Universal Robots PolyScope program: Cover LT.urp

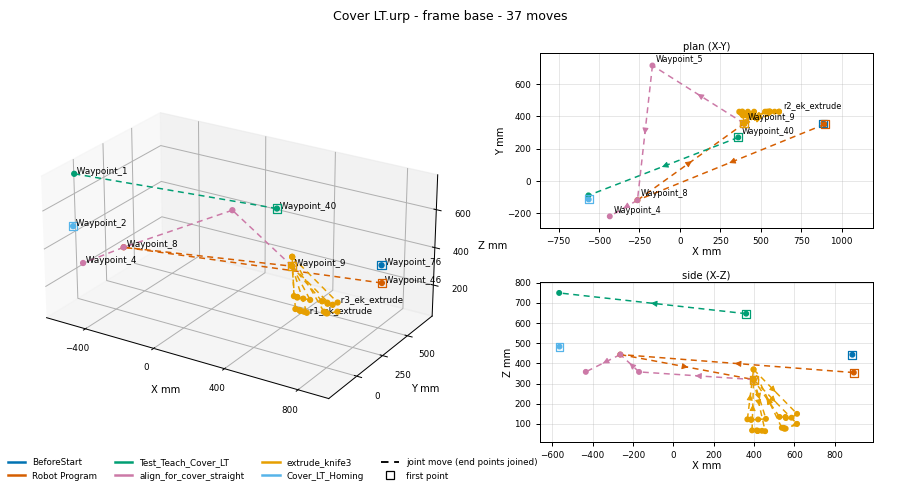
[picture p0: tool path of Cover LT.urp in frame base, 37 of 60 moves have a stored position in this frame; points joined in program order, loops and branches not executed]
Program Cover LT (installation=robot2 directory=/programs/UPF createdIn=5.14.5 lastSavedIn=5.21.3 robotSerialNumber=20246801938)
Calibrated DH parameters: a=[-0.000071, -0.790281, -0.600694, 0.000061, -0.000039, 0]; d=[0.236272, 604.465945, 132.116513, -736.382239, 0.159268, 0.154005]; alpha=[1.570254, -0.000567, 0.000559, 1.571709, -1.56999, 0]; deltaTheta=[0, -0.409357, 7.293326, -0.600784, -0.000001, -0.000001]
InitVariablesNode variables(variable(name=free_dr_already, expression=False), variable(name=freedrive_m_var, expression=False))
BeforeStart
  SuppressedNode
    Folder Safe Home Folder
      'if robot is not at home, send it back to home safely'
      'make sure the tcp is welder'
      Set NoAction tcp=pretend_welder
      sp := get_actual_tcp_pose()
      MoveL speed 250 mm/s, acceleration 1200 mm/s^2 (useActiveTCP=true optimoveEnabled=false optiMoveSpeed=0.3 optiMoveAcceleration=0.09) feature=Base
        Waypoint Variable (Variable): variable=sp
        'if first move is to a variable, skip automove'
      'turn off welder'
      URCap WireTank Serial (WireTank Serial, WireTank, LLC) dataModel(NODE_TITLE=Serial Bridge uR0, Command=[252,82,48], QUERY=false, byte_array=true, OUTPUT_ENTRY=Static, Variable(key=OUTPUT_VARIABLE, variable(name=HwResp)))
      Set DigitalOutput pin=digital_out[0]; digitalValue=0
      jp := get_actual_joint_positions()
      If sp[0]>0.600
        'if x > 600 then above then home'
        MoveJ speed 60 deg/s, acceleration 80 deg/s^2 (useActiveTCP=true optimoveEnabled=false optiMoveSpeed=0.3 optiMoveAcceleration=0.09) feature=Base
          SuppressedNode
            Waypoint Waypoint_47: TCP in base x=894.111 y=351.078 z=354.441 mm, rx=2.3264 ry=2.0525 rz=0.0574 rad; joints [-187.182, -67.293, 94.726, 57.522, -0.141, -88.018] deg; TCP offset x=-5.49 y=-328 z=106.39 mm, rx=1.2092 ry=-1.2092 rz=1.2092 rad
          Waypoint Waypoint_76: TCP in base x=886.939 y=356.263 z=442.999 mm, rx=2.3163 ry=2.0576 rz=0.0741 rad; joints [-187.059, -71.746, 90.665, 52.573, -0.48, -75.13] deg; TCP offset x=-9.5 y=-328 z=105.73 mm, rx=1.2092 ry=-1.2092 rz=1.2092 rad
        SafeHome (positionOptionType=SPEED_AND_ACCELERATION speed=1.047198 acceleration=1.396263 nextMotionTime=2)
      Else 
        Popup Message (haltProgram=false message=retreating to home inputType=Text)
        'for rules 2-8, finish with oldhome then above then home'
        If -1.74<jp[4] and jp[4]<1.05 and -1.74<jp[3] and jp[3]<1.74
          'if oldhome, test teach, then go straight to oldhome'
        ElseIf sp[0]<-.5 and jp[3]>3.14 and -2.62<jp[4] and jp[4]<-0.87
          'if left side weld approach, left weld approach in reverse'
          MoveJ speed 60 deg/s, acceleration 80 deg/s^2 (useActiveTCP=true optimoveEnabled=false optiMoveSpeed=0.3 optiMoveAcceleration=0.09) feature=Base
            Waypoint Waypoint_50: TCP in base x=-568.711 y=230.602 z=220.209 mm, rx=-1.5191 ry=-0.5351 rz=0.574 rad; joints [-1.233, -73.308, 139.365, 291.685, -131.758, 87.871] deg; TCP offset x=-5.49 y=-328 z=106.39 mm, rx=1.2092 ry=-1.2092 rz=1.2092 rad
            Waypoint Waypoint_51: TCP in base x=-689.65 y=139.001 z=230.693 mm, rx=-0.852 ry=-1.646 rz=1.646 rad; joints [-65.631, -88.39, 163.033, 285.278, -280.919, 90.062] deg
            Waypoint Waypoint_52: TCP in base x=-160.992 y=970.528 z=722.037 mm, rx=-0.555 ry=0.1065 rz=0.3285 rad; joints [-74.362, -75.728, 129.393, 212.138, -169.184, 55.164] deg
            Waypoint Waypoint_53: TCP in base x=-157.624 y=513.351 z=815.67 mm, rx=-0.6727 ry=-1.8523 rz=-0.0554 rad; joints [-158.576, -104.315, 132.512, 57.998, -61.68, -46.426] deg
        ElseIf sp[0]<0 and 0<jp[3] and jp[3]<1.74 and 0.87<jp[4] and jp[4]<2.62
          'if right side around, move back then wapoint 24 then oldhome'
          If sp[0]<-1.0
            xback := p[-1.0,sp[1],sp[2],sp[3],sp[4],sp[5]]
            MoveJ speed 60 deg/s, acceleration 80 deg/s^2 (useActiveTCP=true optimoveEnabled=false optiMoveSpeed=0.3 optiMoveAcceleration=0.09) feature=Base
              Waypoint Variable (Variable): variable=xback
          MoveJ speed 60 deg/s, acceleration 80 deg/s^2 (useActiveTCP=true optimoveEnabled=false optiMoveSpeed=0.3 optiMoveAcceleration=0.09) feature=Base
            Waypoint Waypoint_54: TCP in base x=-308.528 y=606.081 z=242.371 mm, rx=-2.1337 ry=0.3494 rz=2.131 rad; joints [-112.4, -74.451, 126.505, 42.726, 91.418, 81.282] deg
        ElseIf jp[3]>2.62 and jp[4]<-3.84
          'if left side second half, then left weld ending sequence'
          If jp[5]<0.35
            MoveJ speed 60 deg/s, acceleration 80 deg/s^2 (useActiveTCP=true optimoveEnabled=false optiMoveSpeed=0.3 optiMoveAcceleration=0.09) feature=Base
              Waypoint Waypoint_65: TCP in base x=-850.3 y=-229.061 z=580.194 mm, rx=-0.0667 ry=-1.5664 rz=-0.0455 rad; joints [6.605, -69.14, 152.414, 186.359, -269.256, -10.612] deg
          MoveJ speed 60 deg/s, acceleration 80 deg/s^2 (useActiveTCP=true optimoveEnabled=false optiMoveSpeed=0.3 optiMoveAcceleration=0.09) feature=Base
            SuppressedNode
              Waypoint Waypoint_61: TCP in base x=-1224.453 y=315.135 z=45.036 mm, rx=0.4556 ry=-1.5209 rz=0.4778 rad; joints [-38.105, -18.537, 102.715, 186.465, -269.531, 72.317] deg
            SuppressedNode
              Waypoint Waypoint_62: TCP in base x=-1246.058 y=121.907 z=25.888 mm, rx=-0.7807 ry=-1.4195 rz=-0.7637 rad; joints [-2.239, -16.844, 100.196, 185.863, -269.635, -54.527] deg
            SuppressedNode
              Waypoint Waypoint_63: TCP in base x=-850.3 y=142.696 z=580.194 mm, rx=-0.0667 ry=-1.5664 rz=-0.0455 rad; joints [-33.715, -70.118, 156.539, 183.763, -269.222, 29.711] deg
            SuppressedNode
              Waypoint Waypoint_64: TCP in base x=-850.307 y=-229.065 z=580.197 mm, rx=-0.0667 ry=-1.5664 rz=-0.0455 rad; joints [6.605, -69.141, 152.414, 186.36, -269.255, -10.612] deg
            'above is testing, below is real'
            Waypoint Waypoint_55: TCP in base x=-850.296 y=369.354 z=580.191 mm, rx=-0.0667 ry=-1.5664 rz=-0.0455 rad; joints [-51.358, -68.674, 149.321, 189.759, -269.326, 47.358] deg
            SuppressedNode
              Waypoint Waypoint_60: TCP in base x=-826.865 y=369.366 z=43.112 mm, rx=0.575 ry=-1.4922 rz=0.5971 rad; joints [-59.177, -17.074, 121.534, 166.294, -269.929, 102.173] deg
            Waypoint Waypoint_59: motionParameters(nextMotionTime=2); TCP in base x=-689.651 y=138.973 z=230.7 mm, rx=-0.852 ry=-1.646 rz=1.646 rad; joints [-65.63, -88.392, 163.034, 285.278, -280.919, 90.062] deg
            Waypoint Waypoint_71: TCP in base x=-289.685 y=534.258 z=757.199 mm, rx=-0.2952 ry=-0.653 rz=0.3894 rad; joints [-79.881, -94.829, 156.624, 238.16, -217.621, 99.184] deg
            Waypoint Waypoint_58: TCP in base x=191.12 y=567.518 z=815.513 mm, rx=-0.1358 ry=0.3961 rz=0.2088 rad; joints [-94.611, -101.484, 149.999, 189.458, -152.19, 49.064] deg
            Waypoint Waypoint_56: TCP in base x=-254.568 y=502.959 z=1135.401 mm, rx=-0.2619 ry=-0.7497 rz=1.3491 rad; joints [-116.567, -108.934, 141.5, 126.12, -66.905, -29.189] deg
            Waypoint Waypoint_57: TCP in base x=-9.221 y=593.713 z=505.809 mm, rx=-1.4244 ry=-2.3441 rz=-0.5276 rad; joints [-167.352, -114.202, 136.688, 39.052, -32.592, -65.93] deg
        ElseIf jp[3]<-2.09
          'bottom homing'
          MoveJ speed 60 deg/s, acceleration 80 deg/s^2 (useActiveTCP=true optimoveEnabled=false optiMoveSpeed=0.3 optiMoveAcceleration=0.09) feature=Base
            SuppressedNode
              Waypoint Waypoint_66: TCP in base x=-1189.333 y=-102.843 z=-176.058 mm, rx=1.1963 ry=-1.1853 rz=1.2301 rad; joints [-19.887, -1.876, 78.341, -165.92, 91.498, 110.543] deg
            ''
            If sp[0]<-0.95
              xback := p[-0.95,sp[1],sp[2],sp[3],sp[4],sp[5]]
              MoveL speed 250 mm/s, acceleration 1200 mm/s^2 (useActiveTCP=true optimoveEnabled=false optiMoveSpeed=0.3 optiMoveAcceleration=0.09) feature=Base
                Waypoint Variable (Variable): variable=xback
            Waypoint Waypoint_67: TCP in base x=-339.169 y=114.271 z=51.007 mm, rx=-0.4342 ry=1.8727 rz=-1.8852 rad; joints [-80.817, -56.025, 141.954, -98.756, -22.671, 103.625] deg
        ElseIf jp[3]<0 and jp[4]<-3.14
          'if left side homing, special unspin'
          MoveJ speed 60 deg/s, acceleration 80 deg/s^2 (useActiveTCP=true optimoveEnabled=false optiMoveSpeed=0.3 optiMoveAcceleration=0.09) feature=Base
            SuppressedNode
              Waypoint Waypoint_68: TCP in base x=-1436.144 y=-207.487 z=20.65 mm, rx=-1.0168 ry=-1.7024 rz=1.6295 rad; joints [2.271, -43.137, 96.498, -42.2, -211.884, 93.908] deg
            ''
            Waypoint Waypoint_69: TCP in base x=-760.827 y=-49.763 z=82.65 mm, rx=-1.0262 ry=-1.6127 rz=1.5471 rad; joints [-12.694, -64.084, 157.914, -89.201, -220.703, 89.352] deg
            Waypoint Waypoint_70: TCP in base x=-154.415 y=636.923 z=16.979 mm, rx=-0.3028 ry=1.487 rz=0.1222 rad; joints [-64.641, -61.184, 139.176, -160.395, -91.873, 99.702] deg
        ElseIf (sp[4]<-3 or sp[4]>3) and -0.02<sp[5] and sp[5]<0.02
          'go straight to home'
        ElseIf 2>1
          'if none of the other options, then error continuously'
          Loop While (checkContinuously=false) expression=2>1
            Popup Message (haltProgram=false message=Unknown Position. Find Calvin for Assistance inputType=Text)
        'insert logic for how to get back to oldhome'
        'finish with oldhome then above then home'
        MoveJ speed 60 deg/s, acceleration 80 deg/s^2 (useActiveTCP=true optimoveEnabled=false optiMoveSpeed=0.3 optiMoveAcceleration=0.09) feature=Base
          Waypoint Waypoint_49: motionParameters(jointSpeed=1.047198 jointAcceleration=1.396263 cartesianSpeed=0.25 cartesianAcceleration=1.2); TCP in base x=397.354 y=356.263 z=319.809 mm, rx=2.3163 ry=2.0576 rz=0.0741 rad; joints [-198.126, -117.851, 133.304, -13.008, -11.424, -6.036] deg
          SuppressedNode
            Waypoint Waypoint_48: TCP in base x=894.09 y=351.09 z=354.453 mm, rx=2.3264 ry=2.0525 rz=0.0573 rad; joints [-187.181, -67.294, 94.727, 57.523, -0.141, -88.018] deg
          Waypoint Waypoint_75: TCP in base x=886.939 y=356.263 z=442.999 mm, rx=2.3163 ry=2.0576 rz=0.0741 rad; joints [-187.059, -71.746, 90.665, 52.573, -0.48, -75.13] deg; TCP offset x=-9.5 y=-328 z=105.73 mm, rx=1.2092 ry=-1.2092 rz=1.2092 rad
        SafeHome (positionOptionType=SPEED_AND_ACCELERATION speed=1.047198 acceleration=1.396263 nextMotionTime=2)
      SuppressedNode
        URCap MachineLogic for Universal Robots (MachineLogic for Universal Robots, Vention Inc.) dataModel(type=addMotor, numberAdded=0, speed_in_mm_per_min=600, acceleration_in_mm_per_s2=50.0, teachColor=BLUE, combo1=MachineMotion1, combo2=(1) Custom Actuator, combo3=Home, combo6=In series, message=Homing, description=Moves the actuator in the negative direction until the home sensor is triggered and sets position to zero (0)., comboAddress=Address 1, comboActuator=Valve 1)
  'for this, dont have to worry about the normal stuff. just send it up and home'
  Folder Cover Safe Home Folder
    'if robot is not at home, send it back to home safely'
    'make sure the tcp is welder'
    Set NoAction tcp=pretend_welder
    sp := get_actual_tcp_pose()
    MoveL speed 250 mm/s, acceleration 1200 mm/s^2 (useActiveTCP=true optimoveEnabled=false optiMoveSpeed=0.3 optiMoveAcceleration=0.09) feature=Base
      Waypoint Variable (Variable): variable=sp
      'if first move is to a variable, skip automove'
    'turn off welder'
    URCap WireTank Serial (WireTank Serial, WireTank, LLC) dataModel(NODE_TITLE=Serial Bridge uR0, Command=[252,82,48], byte_array=true, OUTPUT_ENTRY=Static, QUERY=false, Variable(key=OUTPUT_VARIABLE, variable(name=HwResp)))
    Set DigitalOutput pin=digital_out[0]; digitalValue=0
    jp := get_actual_joint_positions()
    If sp[0]>0.600
      'if x > 600 then above then home'
      MoveJ speed 60 deg/s, acceleration 80 deg/s^2 (useActiveTCP=true optimoveEnabled=false optiMoveSpeed=0.3 optiMoveAcceleration=0.09) feature=Base
        SuppressedNode
          Waypoint Waypoint_47: TCP in base x=894.111 y=351.078 z=354.441 mm, rx=2.3264 ry=2.0525 rz=0.0574 rad; joints [-187.182, -67.293, 94.726, 57.522, -0.141, -88.018] deg; TCP offset x=-5.49 y=-328 z=106.39 mm, rx=1.2092 ry=-1.2092 rz=1.2092 rad
        Waypoint Waypoint_76: TCP in base x=886.939 y=356.263 z=442.999 mm, rx=2.3163 ry=2.0576 rz=0.0741 rad; joints [-187.059, -71.746, 90.665, 52.573, -0.48, -75.13] deg; TCP offset x=-9.5 y=-328 z=105.73 mm, rx=1.2092 ry=-1.2092 rz=1.2092 rad
      SafeHome (positionOptionType=SPEED_AND_ACCELERATION speed=1.047198 acceleration=1.396263 nextMotionTime=2)
    Else 
      Popup Message (haltProgram=false message=retreating to home inputType=Text)
      MoveL speed 250 mm/s, acceleration 1200 mm/s^2 (useActiveTCP=true optimoveEnabled=false optiMoveSpeed=0.3 optiMoveAcceleration=0.09) feature=Base
        MoveDirectionNode (selectedDirection=ZPlus)
          Until DISTANCE (allowActions=false deceleration=3 distanceNodeType=STOP) Distance=0.1; motionParameters(blendRadius=0)
      SuppressedNode
        'for rules 2-8, finish with oldhome then above then home'
      SuppressedNode
        If -1.74<jp[4] and jp[4]<1.05 and -1.74<jp[3] and jp[3]<1.74 removedSiblings(If(type=ElseIf checkContinuously=false, expression=sp[0]<-.5 and jp[3]>3.14 and -2.62<jp[4] and jp[4]<-0.87, children(Comment(comment=if left side weld approach, left weld approach in reverse), Move(motionType=MoveJ speed=1.047198 acceleration=1.396263 useActiveTCP=true positionType=CartesianPose optimoveEnabled=false optiMoveSpeed=0.3 optiMoveAcceleration=0.09, feature=Base, children(Waypoint(type=Fixed name=Waypoint_50, position(JointAngles=[-0.021522, -1.279472, 2.432382, 5.090871, -2.299611, 1.533644], TCPOffset=[-0.00549, -0.328, 0.10639, 1.2092, -1.2092, 1.2092]), BaseToFeature=[0, 0, 0, 0, 0, 0]), Waypoint(type=Fixed name=Waypoint_51, position(JointAngles=[-1.145481, -1.542704, 2.84547, 4.979048, -4.902958, 1.571883], TCPOffset=[-0.00549, -0.328, 0.10639, 1.2092, -1.2092, 1.2092]), BaseToFeature=[0, 0, 0, 0, 0, 0]), Waypoint(type=Fixed name=Waypoint_52, position(JointAngles=[-1.297858, -1.3217, 2.258328, 3.702513, -2.952825, 0.962794], TCPOffset=[-0.00549, -0.328, 0.10639, 1.2092, -1.2092, 1.2092]), BaseToFeature=[0, 0, 0, 0, 0, 0]), Waypoint(type=Fixed name=Waypoint_53, position(JointAngles=[-2.767666, -1.820643, 2.312763, 1.012255, -1.076523, -0.810283], TCPOffset=[-0.00549, -0.328, 0.10639, 1.2092, -1.2092, 1.2092]), BaseToFeature=[0, 0, 0, 0, 0, 0]))))), If(type=ElseIf checkContinuously=false, expression=sp[0]<0 and 0<jp[3] and jp[3]<1.74 and 0.87<jp[4] and jp[4]<2.62, children(Comment(comment=if right side around, move back then wapoint 24 then oldhome), If(type=If checkContinuously=false, expression=sp[0]<-1.0, children(Assignment(valueSource=Expression, variable=xback, expression=p[-1.0,sp[1],sp[2],sp[3],sp[4],sp[5]]), Move(motionType=MoveJ speed=1.047198 acceleration=1.396263 useActiveTCP=true positionType=CartesianPose optimoveEnabled=false optiMoveSpeed=0.3 optiMoveAcceleration=0.09, feature=Base, children(Waypoint(type=Variable name=Variable, variable=xback))))), Move(motionType=MoveJ speed=1.047198 acceleration=1.396263 useActiveTCP=true positionType=CartesianPose optimoveEnabled=false optiMoveSpeed=0.3 optiMoveAcceleration=0.09, feature=Base, children(Waypoint(type=Fixed name=Waypoint_54, position(JointAngles=[-1.961751, -1.299423, 2.207935, 0.745709, 1.59555, 1.418632], TCPOffset=[-0.00549, -0.328, 0.10639, 1.2092, -1.2092, 1.2092]), BaseToFeature=[0, 0, 0, 0, 0, 0]))))), If(type=ElseIf checkContinuously=false, expression=jp[3]>2.62 and jp[4]<-3.84, children(Comment(comment=if left side second half, then left weld ending sequence), If(type=If checkContinuously=false, expression=jp[5]<0.35, children(Move(motionType=MoveJ speed=1.047198 acceleration=1.396263 useActiveTCP=true positionType=CartesianPose optimoveEnabled=false optiMoveSpeed=0.3 optiMoveAcceleration=0.09, feature=Base, children(Waypoint(type=Fixed name=Waypoint_65, position(JointAngles=[0.115278, -1.206729, 2.660133, 3.252583, -4.699399, -0.185216], TCPOffset=[-0.00549, -0.328, 0.10639, 1.2092, -1.2092, 1.2092]), BaseToFeature=[0, 0, 0, 0, 0, 0]))))), Move(motionType=MoveJ speed=1.047198 acceleration=1.396263 useActiveTCP=true positionType=CartesianPose optimoveEnabled=false optiMoveSpeed=0.3 optiMoveAcceleration=0.09, feature=Base, children(SuppressedNode(suppressedNode(type=Fixed name=Waypoint_61, position(JointAngles=[-0.665049, -0.323534, 1.792719, 3.254424, -4.7042, 1.262177], TCPOffset=[-0.00549, -0.328, 0.10639, 1.2092, -1.2092, 1.2092]), BaseToFeature=[0, 0, 0, 0, 0, 0])), SuppressedNode(suppressedNode(type=Fixed name=Waypoint_62, position(JointAngles=[-0.039081, -0.293979, 1.748757, 3.243919, -4.706024, -0.951676], TCPOffset=[-0.00549, -0.328, 0.10639, 1.2092, -1.2092, 1.2092]), BaseToFeature=[0, 0, 0, 0, 0, 0])), SuppressedNode(suppressedNode(type=Fixed name=Waypoint_63, position(JointAngles=[-0.58843, -1.223785, 2.732112, 3.207264, -4.698814, 0.518554], TCPOffset=[-0.00549, -0.328, 0.10639, 1.2092, -1.2092, 1.2092]), BaseToFeature=[0, 0, 0, 0, 0, 0])), SuppressedNode(suppressedNode(type=Fixed name=Waypoint_64, position(JointAngles=[0.115283, -1.206735, 2.660121, 3.252601, -4.699394, -0.185216], TCPOffset=[-0.00549, -0.328, 0.10639, 1.2092, -1.2092, 1.2092]), BaseToFeature=[0, 0, 0, 0, 0, 0])), Comment(comment=above is testing, below is real), Waypoint(type=Fixed name=Waypoint_55, position(JointAngles=[-0.896367, -1.198587, 2.606137, 3.311917, -4.700617, 0.826545], TCPOffset=[-0.00549, -0.328, 0.10639, 1.2092, -1.2092, 1.2092]), BaseToFeature=[0, 0, 0, 0, 0, 0]), SuppressedNode(suppressedNode(type=Fixed name=Waypoint_60, position(JointAngles=[-1.032829, -0.298001, 2.121174, 2.902384, -4.711147, 1.783251], TCPOffset=[-0.00549, -0.328, 0.10639, 1.2092, -1.2092, 1.2092]), BaseToFeature=[0, 0, 0, 0, 0, 0])), Waypoint(type=Fixed name=Waypoint_59, motionParameters(nextMotionTime=2), position(JointAngles=[-1.145453, -1.542729, 2.84548, 4.979044, -4.902961, 1.571883], TCPOffset=[-0.00549, -0.328, 0.10639, 1.2092, -1.2092, 1.2092]), BaseToFeature=[0, 0, 0, 0, 0, 0]), Waypoint(type=Fixed name=Waypoint_71, position(JointAngles=[-1.394185, -1.655085, 2.733613, 4.156679, -3.798194, 1.731084], TCPOffset=[-0.00549, -0.328, 0.10639, 1.2092, -1.2092, 1.2092]), BaseToFeature=[0, 0, 0, 0, 0, 0]), Waypoint(type=Fixed name=Waypoint_58, position(JointAngles=[-1.651281, -1.771235, 2.617982, 3.30666, -2.656208, 0.856331], TCPOffset=[-0.00549, -0.328, 0.10639, 1.2092, -1.2092, 1.2092]), BaseToFeature=[0, 0, 0, 0, 0, 0]), Waypoint(type=Fixed name=Waypoint_56, position(JointAngles=[-2.034486, -1.901249, 2.469647, 2.201206, -1.167719, -0.509439], TCPOffset=[-0.00549, -0.328, 0.10639, 1.2092, -1.2092, 1.2092]), BaseToFeature=[0, 0, 0, 0, 0, 0]), Waypoint(type=Fixed name=Waypoint_57, position(JointAngles=[-2.920838, -1.993208, 2.385661, 0.681589, -0.568846, -1.150698], TCPOffset=[-0.00549, -0.328, 0.10639, 1.2092, -1.2092, 1.2092]), BaseToFeature=[0, 0, 0, 0, 0, 0]))))), If(type=ElseIf checkContinuously=false, expression=jp[3]<-2.09, children(Comment(comment=bottom homing), Move(motionType=MoveJ speed=1.047198 acceleration=1.396263 useActiveTCP=true positionType=CartesianPose optimoveEnabled=false optiMoveSpeed=0.3 optiMoveAcceleration=0.09, feature=Base, children(SuppressedNode(suppressedNode(type=Fixed name=Waypoint_66, position(JointAngles=[-0.347097, -0.032738, 1.367305, -2.895854, 1.59695, 1.929343], TCPOffset=[-0.00549, -0.328, 0.10639, 1.2092, -1.2092, 1.2092]), BaseToFeature=[0, 0, 0, 0, 0, 0])), If(type=If checkContinuously=false, expression=sp[0]<-0.95, children(Assignment(valueSource=Expression, variable=xback, expression=p[-0.95,sp[1],sp[2],sp[3],sp[4],sp[5]]), Move(motionType=MoveL speed=0.25 acceleration=1.2 useActiveTCP=true positionType=CartesianPose optimoveEnabled=false optiMoveSpeed=0.3 optiMoveAcceleration=0.09, feature=Base, children(Waypoint(type=Variable name=Variable, variable=xback))))), Waypoint(type=Fixed name=Waypoint_67, position(JointAngles=[-1.410516, -0.977824, 2.47756, -1.723615, -0.395682, 1.808601], TCPOffset=[-0.00549, -0.328, 0.10639, 1.2092, -1.2092, 1.2092]), BaseToFeature=[0, 0, 0, 0, 0, 0]))))), If(type=ElseIf checkContinuously=false, expression=jp[3]<0 and jp[4]<-3.14, children(Comment(comment=if left side homing, special unspin), Move(motionType=MoveJ speed=1.047198 acceleration=1.396263 useActiveTCP=true positionType=CartesianPose optimoveEnabled=false optiMoveSpeed=0.3 optiMoveAcceleration=0.09, feature=Base, children(SuppressedNode(suppressedNode(type=Fixed name=Waypoint_68, position(JointAngles=[0.039635, -0.752881, 1.684208, -0.736535, -3.698072, 1.639011], TCPOffset=[-0.00549, -0.328, 0.10639, 1.2092, -1.2092, 1.2092]), BaseToFeature=[0, 0, 0, 0, 0, 0])), Waypoint(type=Fixed name=Waypoint_69, position(JointAngles=[-0.221546, -1.118469, 2.756124, -1.556857, -3.851988, 1.559481], TCPOffset=[-0.00549, -0.328, 0.10639, 1.2092, -1.2092, 1.2092]), BaseToFeature=[0, 0, 0, 0, 0, 0]), Waypoint(type=Fixed name=Waypoint_70, position(JointAngles=[-1.128192, -1.067859, 2.429081, -2.799421, -1.603484, 1.74012], TCPOffset=[-0.00549, -0.328, 0.10639, 1.2092, -1.2092, 1.2092]), BaseToFeature=[0, 0, 0, 0, 0, 0]))))), If(type=ElseIf checkContinuously=false, expression=(sp[4]<-3 or sp[4]>3) and -0.02<sp[5] and sp[5]<0.02, children(Comment(comment=go straight to home))), If(type=ElseIf checkContinuously=false, expression=2>1, children(Comment(comment=if none of the other options, then error continuously), Loop(type=While checkContinuously=false, expression=2>1, children(Popup(type=Message haltProgram=false message=Unknown Position. Find Calvin for Assistance inputType=Text))))))
          'if oldhome, test teach, then go straight to oldhome'
      'insert logic for how to get back to oldhome'
      'finish with oldhome then above then home'
      SuppressedNode
        MoveJ speed 60 deg/s, acceleration 80 deg/s^2 (useActiveTCP=true optimoveEnabled=false optiMoveSpeed=0.3 optiMoveAcceleration=0.09) feature=Base
          Waypoint Waypoint_49: motionParameters(jointSpeed=1.047198 jointAcceleration=1.396263 cartesianSpeed=0.25 cartesianAcceleration=1.2); TCP in base x=397.354 y=356.263 z=319.809 mm, rx=2.3163 ry=2.0576 rz=0.0741 rad; joints [-198.126, -117.851, 133.304, -13.008, -11.424, -6.036] deg; TCP offset x=-5.49 y=-328 z=106.39 mm, rx=1.2092 ry=-1.2092 rz=1.2092 rad
          SuppressedNode
            Waypoint Waypoint_48: TCP in base x=894.09 y=351.09 z=354.453 mm, rx=2.3264 ry=2.0525 rz=0.0573 rad; joints [-187.181, -67.294, 94.727, 57.523, -0.141, -88.018] deg
          Waypoint Waypoint_75: TCP in base x=886.939 y=356.263 z=442.999 mm, rx=2.3163 ry=2.0576 rz=0.0741 rad; joints [-187.059, -71.746, 90.665, 52.573, -0.48, -75.13] deg; TCP offset x=-9.5 y=-328 z=105.73 mm, rx=1.2092 ry=-1.2092 rz=1.2092 rad
      SafeHome (positionOptionType=SPEED_AND_ACCELERATION speed=1.047198 acceleration=1.396263 nextMotionTime=2)
      Popup Message (haltProgram=false message=home. start program inputType=Text)
    SuppressedNode
      URCap MachineLogic for Universal Robots (MachineLogic for Universal Robots, Vention Inc.) dataModel(type=addMotor, numberAdded=0, speed_in_mm_per_min=600, acceleration_in_mm_per_s2=50.0, teachColor=BLUE, combo1=MachineMotion1, combo2=(1) Custom Actuator, combo3=Home, combo6=In series, message=Homing, description=Moves the actuator in the negative direction until the home sensor is triggered and sets position to zero (0)., comboAddress=Address 1, comboActuator=Valve 1)
Robot Program (runOnlyOnce=true)
  'start of main program'
  Set NoAction tcp=pretend_welder
  SafeHome (positionOptionType=SPEED_AND_ACCELERATION speed=1.047198 acceleration=1.396263 nextMotionTime=2)
  Script file /programs/common_math.script
    | # this file contains math equations and operations, not specific to any one feature
    | 
    | # define pi
    | pi = 3.1415926535
    | 
    | # given 3 points, this finds the plane and its equation
    | # rereturns ax + by + cz + d = 0 in a list of [a, b, c, d]
    | def findplane(p11, p12, p13):
    |     # extract coordinates
    |     x1 = p11[0]
    |     y1 = p11[1]
    |     z1 = p11[2]
    |     x2 = p12[0]
    |     y2 = p12[1]
    |     z2 = p12[2]
    |     x3 = p13[0]
    |     y3 = p13[1]
    |     z3 = p13[2]
    |     # create vectors from the points
    |     v1x = x2-x1
    |     v1y = y2-y1
    |     v1z = z2-z1
    |     v2x = x3-x1
    |     v2y = y3-y1
    |     v2z = z3-z1
    |     #calculate the normal vector using the cross product
    |     nx = v1y*v2z - v1z*v2y # i component
    |     ny = v1z*v2x - v1x*v2z # j component
    |     nz = v1x*v2y - v1y*v2x # k component
    |     # calculate d in the plane equation
    |     d = -1 * (nx*x1 + ny*y1 + nz*z1)
    |     ret = [nx, ny, nz, d]
    |     return ret
    | end
    | 
    | # this function finds the intersection point between two lines in the xy plane
    | # takes 4 arguments: m1, b1, m2, b2
    | # returns a list of [x,y] (the point of intersection)
    | def find_intersection(m1, b1, m2, b2):
    |   # m1x+b1 = m2x+b2
    |   # m1x - m2x = b2 - b1
    |   # x = (b2-b1) / (m1-m2)
    |   x = (b2-b1) / (m1-m2)
    |   y = m1 * x + b1
    |   ret = [x, y]
    |   return ret
    | end
    | 
    | # this function finds the distance between 2 points in 3d space
    | # it takes 6 arguments: x1, y1, z1, x2, y2, z2
    | # it returns a distance
    | def distance_between(x1, y1, z1, x2, y2, z2):
    |   distsquared = (x2-x1)*(x2-x1)+(y2-y1)*(y2-y1)+(z2-z1)*(z2-z1)
    |   dist = sqrt(distsquared)
    |   return dist
    | end
    | 
    | # this function takes a point, a unit vector, and a distance, and adds the distance to the point in the direction of the unit vector (3d space)
    | # it returns a point as a list of coordinates
    | def add_vectordistance_to_point(xi, yi, zi, uvx, uvy, uvz, delta):
    |   xf = xi + uvx * delta
    |   yf = yi + uvy * delta
    |   zf = zi + uvz * delta
    |   ret = [xf, yf, zf]
    |   return ret
    | end
    | 
    | # this function takes two rotation matrices, and multiplies them together, returning one matrix.
    | # all matrices are in the form of a list.
    | # all matrix values have constant values (no variables)
    | def multiply_matrix(matrix1, matrix2):
    |     # retrieve values
    |     a11 = matrix1[0]
    |     a12 = matrix1[1]
    |     a13 = matrix1[2]
    |     a21 = matrix1[3]
    |     a22 = matrix1[4]
    |     a23 = matrix1[5]
    |     a31 = matrix1[6]
    |     a32 = matrix1[7]
    |     a33 = matrix1[8]
    |     b11 = matrix2[0]
    |     b12 = matrix2[1]
    |     b13 = matrix2[2]
    |     b21 = matrix2[3]
    |     b22 = matrix2[4]
    |     b23 = matrix2[5]
    |     b31 = matrix2[6]
    |     b32 = matrix2[7]
    |     b33 = matrix2[8]
    |     #calculate c values
    |     c11 = a11*b11 + a12*b21 + a13*b31
    |     c12 = a11*b12 + a12*b22 + a13*b32
    |     c13 = a11*b13 + a12*b23 + a13*b33
    |     c21 = a21*b11 + a22*b21 + a23*b31
    |     c22 = a21*b12 + a22*b22 + a23*b32
    |     c23 = a21*b13 + a22*b23 + a23*b33
    |     c31 = a31*b11 + a32*b21 + a33*b31
    |     c32 = a31*b12 + a32*b22 + a33*b32
    |     c33 = a31*b13 + a32*b23 + a33*b33
    |     # return resulting matrix
    |     ret = [c11, c12, c13, c21, c22, c23, c31, c32, c33]
    |     return ret
    | end
    | 
    | # this function converts a matrix to axis angle representations
    | # this matrix is usually a resulting matrix (result of matrix multiplication) in normal use, given as a list
    | # returns a list of [rx,ry,rz]
    | def convert_matrix_to_axang(matrix1):
    |     # retrieve values
    |     a11 = matrix1[0]
    |     a12 = matrix1[1]
    |     a13 = matrix1[2]
    |     a21 = matrix1[3]
    |     a22 = matrix1[4]
    |     a23 = matrix1[5]
    |     a31 = matrix1[6]
    |     a32 = matrix1[7]
    |     a33 = matrix1[8]
    | 
    |     # First Half: find the angle
    |     # find the trace
    |     # using the formula: trace = a11 + a22 + a33
    |     trace = a11 + a22 + a33
    |     # find the angle using the formula: trace(matrix) = 1 + 2 cos(angle)
    |     angle = acos((trace - 1.0)/2.0)
    | 
    |     # Second Half: calculate the rotation axis
    |     axisxraw = a32 - a23
    |     axisyraw = a13 - a31
    |     axiszraw = a21 - a12
    |     # normalize axis
    |     magnitude = sqrt(axisxraw*axisxraw + axisyraw*axisyraw + axiszraw*axiszraw)
    |     axisxunit = axisxraw / magnitude
    |     axisyunit = axisyraw / magnitude
    |     axiszunit = axiszraw / magnitude
    | 
    |     # combine axis and angle into rxryrz representation
    |     rxout = axisxunit * angle
    |     ryout = axisyunit * angle
    |     rzout = axiszunit * angle
    |     return [rxout, ryout, rzout]
    | end
    | 
    | # this function takes a rotation and calculates the corresponding rotation matrix
    | # input is (axis, direction, angle in radians)
    | # example is ("x", 1, pi/6) = a 30 degree turn around the x axis in the positive direction (right hand rule)
    | # returns a matrix (a list of 9 values)
    | def get_rotation_matrix_from_description(axis, direction, angle):
    |     # get the angle
    |     a = angle * direction
    |     # get the axis
    |     if axis == "x" or axis == "X":
    |         matrix = [1, 0, 0, 0, cos(a), -1 * sin(a), 0, sin(a), cos(a)]
    |         return matrix
    |     end
    |     if axis == "y" or axis == "Y":
    |         matrix = [cos(a), 0, sin(a), 0, 1, 0, -1*sin(a), 0, cos(a)]
    |         return matrix
    |     end
    |     if axis == "z" or axis == "Z":
    |         matrix = [cos(a), -1*sin(a), 0, sin(a), cos(a), 0, 0, 0, 1]
    |         return matrix
    |     end
    |     # bad
    |     popuptext = "Error in get_rotation_matrix_from_description. "
    |     # infinite loop
    |     while 1==1:
    |       popup(popuptext, title="Code Error",blocking=True)
    |     end
    | end
    | 
    | # given a round over distance (in mm), calculate (based on 90 degrees) the distance from corner (line intersection) to midpoint of arc
    | # returns a value (in mm) that you need to move from line intersection to midpoint (actual distance will be this times sqrt(2))
    | def calc_rod_midpoint_90deg(rod):
    |     # the factor is (1- 1/sqrt(2))
    |     factor = 0.292893
    |     ret = rod * factor
    |     return ret
    | end
    | 
    | def crossproduct(vec1, vec2):
    |     nx = vec1[1]*vec2[2] - vec1[2]*vec2[1]
    |     ny = vec1[2]*vec2[0] - vec1[0]*vec2[2]
    |     nz = vec1[0]*vec2[1] - vec1[1]*vec2[0]
    |     ret = [nx, ny, nz]
    |     return ret
    | end
    | 
    | # Section: headings, angles, slopes conversions
    | 
    | # this function converts a heading (ccw radians from the positive x axis) into rxryrz to be put into a point p[]
    | # this will point the gun in this heading with the bottom side of the gun facing up.
    | # the values used in this program were calculated by doing rotation matrix math in the file on WI-CALVINB10 C. Documents. Theory for converting rotations into axis angle representations
    | def convert_heading_to_axang(heading):
    |  axisxraw = -1 * sin(heading)
    |  axisyraw = cos(heading) + 1
    |  axiszraw = sin(heading)
    | 
    |  magnitude = sqrt(axisxraw*axisxraw + axisyraw*axisyraw + axiszraw*axiszraw)
    | 
    |  axisxunit = axisxraw / magnitude
    |  axisyunit = axisyraw / magnitude
    |  axiszunit = axiszraw / magnitude
    | 
    |  angle = acos( (cos(heading) - 1) / 2 )
    | 
    |  rxout = axisxunit * angle
    |  ryout = axisyunit * angle
    |  rzout = axiszunit * angle
    | 
    |  return [rxout, ryout, rzout]
    | end
    | 
    | # this function converts a heading (ccw radians from the positive x axis) into rxryrz to be put into a point p[]
    | # this will point the gun in this heading with the preheat side of the gun tip facing up. Used for welding in a vertical path.
    | # the values used in this program were calculated by doing rotation matrix math in the file on WI-CALVINB10 C. Documents. Theory for converting rotations into axis angle representations
    | def convert_heading_to_axang_preheatup(heading):
    |  axisxraw = -sin(heading) + 1
    |  axisyraw = cos(heading)
    |  axiszraw = cos(heading)
    | 
    |  magnitude = sqrt(axisxraw*axisxraw + axisyraw*axisyraw + axiszraw*axiszraw)
    | 
    |  axisxunit = axisxraw / magnitude
    |  axisyunit = axisyraw / magnitude
    |  axiszunit = axiszraw / magnitude
    | 
    |  angle = acos( (-sin(heading) - 1) / 2 )
    | 
    |  rxout = axisxunit * angle
    |  ryout = axisyunit * angle
    |  rzout = axiszunit * angle
    | 
    |  return [rxout, ryout, rzout]
    | end
    | 
    | # this function converts a heading (ccw radians from the positive x axis) into rxryrz to be put into a point p[]
    | # this will point the gun in this heading with the preheat side of the gun tip facing down. Used for welding in a vertical path downwards.
    | # the values used in this program were calculated by doing rotation matrix math in the file on WI-CALVINB10 C. Documents. Theory for converting rotations into axis angle representations
    | def convert_heading_to_axang_preheatdown(heading):
    |  axisxraw = -sin(heading) - 1
    |  axisyraw = cos(heading)
    |  axiszraw = -cos(heading)
    | 
    |  magnitude = sqrt(axisxraw*axisxraw + axisyraw*axisyraw + axiszraw*axiszraw)
    | 
    |  axisxunit = axisxraw / magnitude
    |  axisyunit = axisyraw / magnitude
    |  axiszunit = axiszraw / magnitude
    | 
    |  angle = acos( (sin(heading) - 1) / 2 )
    | 
    |  rxout = axisxunit * angle
    |  ryout = axisyunit * angle
    |  rzout = axiszunit * angle
    | 
    |  return [rxout, ryout, rzout]
    | end
    | 
    | # this function converts a heading (ccw radians from the positive x axis) into rxryrz to be put into a point p[]
    | # this will point the gun in this heading with the preheat side of the gun tip facing right. Used for welding counterclockwise around the box.
    | # the values used in this program were calculated by doing rotation matrix math in the file on WI-CALVINB10 C. Documents. Theory for converting rotations into axis angle representations
    | def convert_heading_to_axang_ccw(heading):
    |  axisxraw = -sin(heading)
    |  axisyraw = cos(heading) - 1
    |  axiszraw = -sin(heading)
    | 
    |  magnitude = sqrt(axisxraw*axisxraw + axisyraw*axisyraw + axiszraw*axiszraw)
    | 
    |  axisxunit = axisxraw / magnitude
    |  axisyunit = axisyraw / magnitude
    |  axiszunit = axiszraw / magnitude
    | 
    |  angle = acos( (-cos(heading) - 1) / 2 )
    | 
    |  rxout = axisxunit * angle
    |  ryout = axisyunit * angle
    |  rzout = axiszunit * angle
    | 
    |  return [rxout, ryout, rzout]
    | end
    | 
    | # given a heading, (ccw from +x axis), find the mx+b slope
    | # fails if exactly vertical
    | def get_slope_from_heading(heading):
    |     return tan(heading)
    | end
    | 
    | # this function converts a unit vector to its heading angle ccw from x+ axis
    | # takes uvx and uvy
    | # returns heading in radians
    | def convert_uv_to_heading(uvx, uvy):
    |   baseang = atan(uvy/uvx)
    |   if uvx < 0:
    |     ang = baseang + pi
    |   elif uvy < 0:
    |     ang = baseang + pi * 2
    |   else:
    |     ang = baseang
    |   end
    |   return ang
    | end
    | 
    | # this function finds the equation of a line, perpendicular to a given line, and going through a given point
    | # takes 3 arguments: m (the original line's slope), x (point's x coord), y (point's y coord). the b of the original line is not needed
    | # returns a list of [m,b] (the slope and intercept of the new line)
    | def find_perpendicular_line(origm, x, y):
    |   m = (1/origm) * -1
    |   b = y - m*x
    |   ret = [m, b]
    |   return ret
    | end
    | 
    | # returns the absolute value of a number
    | def absolute(x):
    |     ret = x
    |     if x < 0:
    |         ret = -1 * x
    |     end
    |     return ret
    | end
  Script file /programs/common_io.script
    | # common_io.script
    | # this file contains IO (input/output) commands, commonly used by robot programs
    | # includes rs232 commands, lift column commands, and calls to native universal robots functions (like get_inverse_kin_has_solution())
    | 
    | 
    | # Section: rs232 commands ###############################
    | 
    | # this function sends a signal to turn extrusion on
    | def turn_extrusion_on():
    |   # flush the channel
    |   resp0 = send_serial_signal(["u", "r", "?"])
    |   # send the signal
    |   resp1 = send_serial_signal(["u", "R", "1"])
    |   # if resp <> "uR1"
    |   if resp1 != [252,82,49]:
    |     # turn off extrusion and heating. inform calvin
    |     resp2 = send_serial_signal(["u", "R", "0"])
    |     resp3 = send_serial_signal(["u", "H", "0"])
    |     popuptext = "Error code encountered while trying to start extrusion. Find Calvin. "
    |     while 1==1:
    |       popup(popuptext, title="Extrusion Error Code",blocking=True)
    |       popup(resp1, blocking=True)
    |     end
    |   end
    | end
    | 
    | # this function sends a signal and receives a response
    | # signal is a list of 3 strings, 1 character each. first is u. second is the next character. third is final character
    | def send_serial_signal(signal):
    |   signal2char = signal[1]
    |   signal3char = signal[2]
    |   listsignal = [252, get_corr_number(signal2char), get_corr_number(signal3char)]
    |   resp1 = WTSerialBridge.send_command("/dev/ttyUSB0",1200, 8, "None", "One", "None", 1000, "None", "None", listsignal, True)
    |   return resp1
    | end
    | 
    | # this function converts a letter into its ascii number
    | def get_corr_number(letter):
    |   if letter == "A":
    |     return 65
    |   elif letter == "H":
    |     return 72
    |   elif letter == "R":
    |     return 82
    |   elif letter == "M":
    |     return 77
    |   elif letter == "E":
    |     return 69
    |   elif letter == "a":
    |     return 97
    |   elif letter == "b":
    |     return 98
    |   elif letter == "h":
    |     return 104
    |   elif letter == "r":
    |     return 114
    |   elif letter == "s":
    |     return 115
    |   elif letter == "m":
    |     return 109
    |   elif letter == "0":
    |     return 48
    |   elif letter == "1":
    |     return 49
    |   elif letter == "2":
    |     return 50
    |   elif letter == "3":
    |     return 51
    |   elif letter == "4":
    |     return 52
    |   elif letter == "5":
    |     return 53
    |   elif letter == "6":
    |     return 54
    |   elif letter == "7":
    |     return 55
    |   elif letter == "8":
    |     return 56
    |   elif letter == "9":
    |     return 57
    |   elif letter == "?":
    |     return 63
    |   end
    | end
    | 
    | # this function checks whether the welder is in the ready state.
    | # to be called at the beginning of Main Program
    | def welder_state_ready():
    |   # flush the channel
    |   resp0 = send_serial_signal(["u", "s", "?"])
    |   # send the signal
    |   resp1 = send_serial_signal(["u", "s", "?"])
    |   # if resp1 == [252,115,49] (us1) then it is ready. otherwise, it is not
    |   if resp1 != [252,115,49]:
    |     popuptext = "Welder is not ready for extrusion. Follow the instructions to start heating welder. "
    |     while 1==1:
    |       popup(popuptext, title="Welder Not Ready",blocking=True)
    |     end
    |   end
    | 
    | end
    | 
    | 
    | # Section: lift column commands ##################################
    | 
    | # initialize a lift column extension needed of 0.0
    | global liftcolumnzneeded = 0.0 # set this variable in mm
    | 
    | def get_lift_column_height():
    |   # begin: URCap Program Node
    |   #   Source: MachineLogic for Universal Robots, 3.1.7, Vention Inc.
    |   #   Type: MachineLogic for Universal Robots
    |   #$ 5 "MachineLogic Get Position"
    |   while isVentionMovementBusyMachineMotion1==True:
    |     sleep(0.05)
    |   end
    |   if(isVentionMovementBusyMachineMotion1 == False):
    |     isVentionMovementBusyMachineMotion1 = True
    |     socket_send_string("estop/status;", "MachineMotion1")
    |     temp_estop_var_vention = socket_read_string("MachineMotion1",timeout=15)
    |     while(temp_estop_var_vention=="estop/status true"):
    |       if temp_estop_var_vention=="estop/status true":
    |         sendStringWithTimeout("estop/systemreset/request","Ack estop/systemreset/request;","MachineMotion1")
    |       end
    |       socket_send_string("estop/status;", "MachineMotion1")
    |       temp_estop_var_vention = socket_read_string("MachineMotion1",timeout=15)
    |       if temp_estop_var_vention=="estop/status true":
    |         popup("MachineMotion in estop, make sure you have all emergency modules released manually. If you continue the system will try to reset MachineMotion automatically.",blocking=True)
    |       end
    |     end
    |   else:
    |     popup("resource is being used already: MachineMotion1")
    |     halt
    |   end
    |   socket_send_string("GET im_get_controller_pos_axis_1;", "MachineMotion1")
    |   temp_drive = socket_read_ascii_float(1, "MachineMotion1",timeout=15)
    |   global var_1 = temp_drive[1]
    |   isVentionMovementBusyMachineMotion1 = False
    |   sleep(0.03)
    |   # end: URCap Program Node
    | end
    | 
    | 
    | def get_lift_column_height_condensed():
    |   socket_send_string("GET im_get_controller_pos_axis_1;", "MachineMotion1")
    |   temp_drive = socket_read_ascii_float(1, "MachineMotion1",timeout=15)
    |   ret = temp_drive[1]
    |   return ret
    | end
    | 
    | 
    | # Section: Native UR commands ###################################
    | 
    | # this function takes a struct of points as an argument, and checks whether every point in the list is reachable using get_inverse_kin_has_solution()
    | # this function does NOT check for weird twists or joint limits
    | # inputstruct must contain only points
    | # it returns true if all points are valid. it returns false if any points are valid
    | # a list of length 0 indicates that all points are valid
    | def check_structofpoints_validity(inputstruct):
    |   # next, check whether the touchpoints are reachable
    |   structlength = length(inputstruct)
    |   i = 0
    |   allvalid = True
    |   while i < structlength:
    |     curr = inputstruct[i]
    |     valid = get_inverse_kin_has_solution(curr)
    |     if not valid:
    |       return False
    |     end
    |     i = i + 1
    |   end
    |   return True
    | end
    | 
    | 
    | # this function takes in a struct of only points. it checks those points for validity.
    | # if one of them is not valid, it throws a popup loop
    | def check_validity_only(struct2):
    |   validity = check_structofpoints_validity(struct2)
    |   if not validity:
    |     # bad
    |     popuptext = "Not all weldpoints are valid. "
    |     # infinite loop
    |     while 1==1:
    |       popup(popuptext, title="Position Error",blocking=True)
    |     end
    |   end
    | end
    | 
    | 
    | # this function calculates whether a given pose can be reached, and if it can, whether it requires a wrist twist (from the seed joint angles)
    | # arguments are target pose (p[x,y,z,rx,ry,rz]) and orig_joints which is the 6 joint angles of a pose that is close by the target pose and has the desired joint angles
    | # returns true if the pose is valid and requires no twist. If pose is valid but requires a twist, returns false. If pose is invalid, returns false.
    | def can_pose_be_reached_without_twist(pose, orig_joints):
    |   # first, determine if the pose is valid
    |   valid = get_inverse_kin_has_solution(pose)
    |   if not valid:
    |     return False
    |   end
    |   valid = get_inverse_kin_has_solution(pose, orig_joints)
    |   if not valid:
    |     return False
    |   else:
    |     joints_1 = get_inverse_kin(pose, orig_joints)
    |     #iterate through the 6 joints
    |     allGood = True
    |     i = 0
    |     structlength = 6
    |     while i < structlength:
    |       joint_curr = joints_1[i]
    |       # check for anything that exceeds joint limits
    |       degreesmax = 360 * pi / 180
    |       if joint_curr > degreesmax or joint_curr < degreesmax * -1:
    |         allGood = False
    |       end
    |       # check for anything that is significantly different than the aligned approach. could indicate a twist is needed. we dont want that
    |       maxdifference = 150 * pi / 180
    |       difference = joint_curr - orig_joints[i]
    |       if difference > maxdifference or difference * -1 > maxdifference:
    |         allGood = False
    |       end
    |       i = i + 1
    |     end
    |     return allGood
    |   end
    | end
  Script file /programs/analyze_coverlt.script
    | def main_calculate_cover_lt(p11, p12, leftpoint, rightpoint):
    |     struct1 = analyze_touchpoints_only_cover_lt(p11, p12, leftpoint, rightpoint)
    |     struct2 = calculate_points_cover_lt(struct1)
    |     #struct2 = calculate_DOtA_points_left_extended(struct1, list1, chamferover, chamferup, tcp_pose_top)
    |     #struct3 = check_validity_left(struct1, struct2)
    |     return struct2
    | 
    | end
    | 
    | def analyze_touchpoints_only_cover_lt(p11, p12, leftpoint, rightpoint):
    |     # calculate the slope of the groove in xy plane
    |     l1p1x = leftpoint[0]
    |     l1p1y = leftpoint[1]
    |     l1p2x = rightpoint[0]
    |     l1p2y = rightpoint[1]
    | 
    |     # equate the first line in 2d space
    |     ml1 = (l1p2y-l1p1y) / (l1p2x-l1p1x)
    | 
    |     # b = y - mx
    |     bl1 = l1p1y - ml1 * l1p1x
    | 
    |     # zraise (how much the z value changes from left point to right point
    |     zraise = p12[2] - p11[2]
    | 
    |     #get the calcpoints
    |     leftcalcpoint = [leftpoint[0], leftpoint[1], p11[2]]
    |     rightcalcpoint = [rightpoint[0], rightpoint[1], p12[2]]
    |     # get the vector from a to b
    |     vec = [rightcalcpoint[0] - leftcalcpoint[0], rightcalcpoint[1] - leftcalcpoint[1], rightcalcpoint[2] - leftcalcpoint[2]]
    |     # get the unit vector in 3d
    |     mag3d = sqrt(vec[0]*vec[0]+vec[1]*vec[1]+vec[2]*vec[2])
    |     vec3dunit = [vec[0]/mag3d, vec[1]/mag3d, vec[2]/mag3d]
    |     # get the unit vector in 2d
    |     mag2d = sqrt(vec[0]*vec[0]+vec[1]*vec[1])
    |     vec2dunit = [vec[0]/mag2d, vec[1]/mag2d]
    |     # get the heading
    |     heading1 = convert_uv_to_heading(vec2dunit[0], vec2dunit[1])
    | 
    |     ret = struct(leftcalcpoint=leftcalcpoint, rightcalcpoint=rightcalcpoint, vxunit=vec3dunit[0], vyunit=vec3dunit[1], vzunit=vec3dunit[2], heading1=heading1)
    |     return ret
    | end
    | 
    | # based on the analysis, calculates the weld path points for the ltude welds.
    | # returns a struct of the weld path points.
    | def calculate_points_cover_lt(struct1):
    |     # get the stuff from struct
    |     leftcalcpoint = struct1[0]
    |     x = leftcalcpoint[0]
    |     y = leftcalcpoint[1]
    |     z = leftcalcpoint[2]
    |     rightcalcpoint = struct1[1]
    |     x2 = rightcalcpoint[0]
    |     y2 = rightcalcpoint[1]
    |     z2 = rightcalcpoint[2]
    |     v3xunit = struct1[2]
    |     v3yunit = struct1[3]
    |     v3zunit = struct1[4]
    |     heading1 = struct1[5]
    | 
    |     # first calculate rxryrz f normal and tiltback
    |     # calculate rxryrz for tilted back
    |     # 3 rotations to make this happen.
    |     # start point is straight up with the preheat pointed in the +y direction.
    |     # first rotation is 180 degrees about x direction. gun is now pointing straight down with preheat facing -y direction
    |     m1 = get_rotation_matrix_from_description("x", 1, 180 * pi / 180)
    |     # second rotation is a 10 degree turn about the x axis (negative direction)
    |     m2 = get_rotation_matrix_from_description("x", -1, 10 * pi / 180)
    |     # third rotation is about 180 degrees about the z axis. starting from the -y axis, go until you get to heading1. that will equal heading1 plus 90 degrees
    |     m3 = get_rotation_matrix_from_description("z", 1, pi/2 + heading1)
    |     # combine them by multiplying m3 * m2 * m1
    |     # matrix multiplication is not commutative but it IS associative, so you can do this whichever order
    |     m4 = multiply_matrix(m2, m1)
    |     m5 = multiply_matrix(m3, m4)
    |     rxryrzt = convert_matrix_to_axang(m5)
    |     rxt = rxryrzt[0]
    |     ryt = rxryrzt[1]
    |     rzt = rxryrzt[2]
    | 
    |     # calculate rxryrz for nontilted
    |     # first rotation is 180 degrees about x direction. gun is now pointing straight down with preheat facing -y direction
    |     m1 = get_rotation_matrix_from_description("x", 1, 180 * pi / 180)
    |     # third rotation is about 180 degrees about the z axis. starting from the -y axis, go until you get to heading1. that will equal heading1 plus 90 degrees
    |     m3 = get_rotation_matrix_from_description("z", 1, pi/2 + heading1)
    |     m5 = multiply_matrix(m3, m1)
    |     rxryrz = convert_matrix_to_axang(m5)
    |     rx = rxryrz[0]
    |     ry = rxryrz[1]
    |     rz = rxryrz[2]
    | 
    |     tiltraise = 0.006 # 6 mm raise needed for the tip to clear the plane during tiltback
    | 
    |     # calculate points 1-3
    |     # calculate point1 (preheat)
    |     dist = -1 * 25.4 / 1000.0 # move back 1 inch from
    |     p1x = x + dist * v3xunit
    |     p1y = y + dist * v3yunit
    |     p1z = z + dist * v3zunit + tiltraise
    |     point1 = p[p1x, p1y, p1z, rxt, ryt, rzt]
    | 
    |     # calculate point2 (start of flatten)
    |     dist = 0.5 * 25.4 / 1000.0  # half an inch past the top of v chamfer
    |     p2x = x + dist * v3xunit
    |     p2y = y + dist * v3yunit
    |     p2z = z + dist * v3zunit + tiltraise
    |     point2 = p[p2x, p2y, p2z, rxt, ryt, rzt]
    | 
    |     # calculate point3 (end of flatten)
    |     dist = 1.5 * 25.4 / 1000.0  # 1.5 inches past top of v chamfer
    |     p3x = x + dist * v3xunit
    |     p3y = y + dist * v3yunit
    |     p3z = z + dist * v3zunit
    |     point3 = p[p3x, p3y, p3z, rx, ry, rz]
    | 
    |     # calculate points 4-6
    |     # calculate point4 (start of unflatten)
    |     dist = -1.5 * 25.4 / 1000.0
    |     p4x = x2 + v3xunit * dist
    |     p4y = y2 + v3yunit * dist
    |     p4z = z2 + v3zunit * dist
    |     point4 = p[p4x, p4y, p4z, rx, ry, rz]
    | 
    |     # calculate point5 (end of unflatten)
    |     dist = -0.5 * 25.4 / 1000.0
    |     p5x = x2 + v3xunit * dist
    |     p5y = y2 + v3yunit * dist
    |     p5z = z2 + v3zunit * dist + tiltraise
    |     point5 = p[p5x, p5y, p5z, rxt, ryt, rzt]
    | 
    |     # calculate point6 (end of smear)
    |     dist = 2 * 25.4 / 1000.0
    |     p6x = x2 + v3xunit * dist
    |     p6y = y2 + v3yunit * dist
    |     p6z = z2 + v3zunit * dist + tiltraise
    |     point6 = p[p6x, p6y, p6z, rxt, ryt, rzt]
    | 
    |     # return struct
    |     ret = struct(point1=point1, point2=point2, point3=point3, point4=point4, point5=point5, point6=point6)
    |     return ret
    | 
    | end
    | 
    | 
    | # this function determines the starting touchpoints for homing in on cover lt geometry
    | # includes two points above the cover lt, closer to the robot than the lt, facing down
    | def get_coverlt_homing_pathpoints(leftpoint, rightpoint):
    |     # get the teach position points
    |     lpx = leftpoint[0]
    |     lpy = leftpoint[1]
    |     lpz = leftpoint[2]
    |     rpx = rightpoint[0]
    |     rpy = rightpoint[1]
    |     rpz = rightpoint[2]
    | 
    |     # determine if the points are parallel (to the tank) or perpendicular
    |     xdelt = absolute(lpx - rpx)
    |     ydelt = absolute(lpy - rpy)
    |     xvcut = False
    |     if xdelt > ydelt:
    |         xvcut = True
    |     end
    | 
    |     # specify the distances from (in meters)
    |     d0 = 0.05 # how far from the cover to approach from
    |     d1 = 0.03 # how far the touchpoints are pushed closer to the robot, offset from the groove
    |     d2 = 0.00 # how far inwards the touchpoints are pushed
    | 
    |     # rxryrz of left point (point 1, taken second): preheat back towards robot to avoid collision with divider wall
    |     rxryrz = [2.014, -2.411, 0]
    |     rx = rxryrz[0]
    |     ry = rxryrz[1]
    |     rz = rxryrz[2]
    | 
    |     # calculate the points
    |     ph1 = p[lpx + d1, lpy + d2, lpz + d0, rx, ry, rz] # left side approach
    |     if xvcut:
    |         ph1 = p[lpx, lpy - d1, lpz + d0, rx, ry, rz] # left side approach
    |     end
    | 
    |     # rxryrz of right point (point 2, taken first): preheat to the left (front) of the tank.
    |     rxryrz2 = [0.334, 3.124, 0]
    |     rx2 = rxryrz2[0]
    |     ry2 = rxryrz2[1]
    |     rz2 = rxryrz2[2]
    | 
    |     ph2 = p[rpx + d1, rpy - d2, rpz + d0, rx2, ry2, rz2] # right side approach
    |     if xvcut:
    |         ph2 = p[rpx, rpy - d1, rpz + d0, rx2, ry2, rz2] # right side approach
    |     end
    | 
    |     ret = struct(ph1=ph1, ph2=ph2)
    |     check_validity_only(ret)
    |     return ret
    | end
    | 
    | # this function runs after the two points have been taught for cover lt. it checks whether the weld points for this line are reachable.
    | # it returns a true or false
    | def check_points_reachable(leftpoint, rightpoint):
    |     struct1t = analyze_touchpoints_only_cover_lt(leftpoint, rightpoint, leftpoint, rightpoint) # use the z of the actual teach point just for checking
    |     points = calculate_points_cover_lt(struct1t)
    |     allvalid = check_structofpoints_validity(points)
    |     if not allvalid:
    |         return False
    |     end
    | 
    |     # now that they are all valid, check if there are any weird turns
    |     # what are the normal joint positions of a regular LT weld?
    |     # left to right: actually left to right and front to back have the same criteria for valid.
    |     # need to get the pre-point
    |     wayp7 = p[-.262598515057, -.117910587405, .443766749060, .115341915577, 3.114598670938, .265717910023]
    |     wayp7q = [0.09593799853302087, -2.4789207352067226, 2.256866488629104, 0.22882056286890795, 1.7417236956390747, -0.16791597406715297]
    |     wayp4 = p[-.433664641517, -.217871332139, .358001604360, -1.895549759225, 2.498965706218, .036945701764]
    |     wayp4q = [-0.6685436407672327, -2.098424097100729, 2.2798998991595667, -0.2272131007960816, -0.39710790315736944, 0.02628905698657036]
    |     if is_xvcut(leftpoint, rightpoint):
    |         prev = wayp4q
    |     else:
    |         prev = wayp7q
    |     end
    |     structlength = 6 # length of points
    |     #listpointnames
    |     lpn = ["p1","p2","p3","p4","p5","p6"]
    |     #pretend_welder_tcp
    |     pwt = p[-0.0117, -0.328, 0.105, 1.2092, -1.2092, 1.2092]
    |     i = 0
    |     while i < structlength:
    |         curr = points[i]
    |         # test this point for nontwist
    |         joints_1 = get_inverse_kin(curr, prev, tcp=pwt)
    |         shoulder = joints_1[1]
    |         if shoulder > 0:
    |             popuptext = "shoulder point " + lpn[i]
    |             popup(popuptext, title="Position Error", blocking=True)
    |             return False
    |         end
    |         elbow = joints_1[2]
    |         if elbow < 0:
    |             popuptext = "elbow point " + lpn[i]
    |             popup(popuptext, title="Position Error", blocking=True)
    |             return False
    |         end
    |         wrist1 = joints_1[3] * 180/pi
    |         if ((wrist1 < -200) or (wrist1 > 100)):
    |             popuptext = "wrist1 point " + lpn[i]
    |             popup(popuptext, title="Position Error", blocking=True)
    |             return False
    |         end
    |         wrist3 = joints_1[5] * 180/pi
    |         if ((wrist3 < -100) or (wrist3 > 100)):
    |             popuptext = "wrist3 point " + lpn[i]
    |             popup(popuptext, title="Position Error", blocking=True)
    |             return False
    |         end
    |         # end of loop
    |         prev = joints_1
    |         i = i + 1
    |     end
    | 
    |     return allvalid
    | end
    | 
    | def is_xvcut(leftpoint, rightpoint):
    |     # get the teach position points
    |     lpx = leftpoint[0]
    |     lpy = leftpoint[1]
    |     lpz = leftpoint[2]
    |     rpx = rightpoint[0]
    |     rpy = rightpoint[1]
    |     rpz = rightpoint[2]
    | 
    |     # determine if the points are parallel (to the tank) or perpendicular
    |     xdelt = absolute(lpx - rpx)
    |     ydelt = absolute(lpy - rpy)
    |     xvcut = False
    |     if xdelt > ydelt:
    |         xvcut = True
    |     end
    |     return xvcut
    | end
  SuppressedNode
    Script: welder_state_ready()
  SuppressedNode
    sidewallchoice :=  (valueSource=Operator message=Is the sidewall 3/4 inch? valueType=Boolean)
  SuppressedNode
    If sidewallchoice removedSiblings(If(type=Else checkContinuously=false, children(Assignment(valueSource=Expression, variable(name=sidewall), expression=0.375))))
      sidewall := 0.628
  SuppressedNode
    deepcham :=  (valueSource=Operator message=Is the chamfer extra deep? (more than 0.21) valueType=Boolean)
  MoveJ speed 60 deg/s, acceleration 80 deg/s^2 (useActiveTCP=true positionType=JointAngles optimoveEnabled=false optiMoveSpeed=0.3 optiMoveAcceleration=0.09) feature=Base
    Waypoint Waypoint_46: TCP in base x=894.108 y=351.078 z=354.456 mm, rx=2.3264 ry=2.0525 rz=0.0574 rad; joints [-187.182, -67.294, 94.726, 57.522, -0.141, -88.018] deg; TCP offset x=-5.49 y=-328 z=106.39 mm, rx=1.2092 ry=-1.2092 rz=1.2092 rad
  Set NoAction tcp=pretend_w_top
  Script: Test_Teach_Cover_LT()
  Folder check validity
    'check validity'
    valid := check_points_reachable(tcp_pose_left,tcp_pose_right)
    SuppressedNode
      If not valid
        Loop Forever
          Popup Message (haltProgram=false message=cannot reach. stop program and retry inputType=Text)
  Set NoAction tcp=pretend_w_top
  Script: kill threadId_Thread_1
  Script: Cover_LT_Homing()
  Set NoAction tcp=pretend_welder
  SuppressedNode
    path1 := analyze_touchpoints(p11,p12,p21,p22,p3)
  SuppressedNode
    CallSubProgram
  SuppressedNode
    MoveJ speed 60 deg/s, acceleration 80 deg/s^2 (useActiveTCP=true optimoveEnabled=false optiMoveSpeed=0.3 optiMoveAcceleration=0.09) feature=Base
      Waypoint Waypoint_19: TCP in base x=-539.433 y=254.004 z=21.521 mm, rx=-1.7232 ry=0.9213 rz=1.7071 rad; joints [-41.97, -63.602, 146.502, 9.159, 84.533, 189.272] deg; TCP offset x=8.55 y=-271.52 z=102 mm, rx=1.2092 ry=-1.2092 rz=1.2092 rad
  pathturn := main_calculate_cover_lt(p11,p12, tcp_pose_left, tcp_pose_right)
  Folder extrude knife
    lch := get_lift_column_height_condensed()
    If lch > 1
      URCap MachineLogic for Universal Robots (MachineLogic for Universal Robots, Vention Inc.) dataModel(type=addMotor, numberAdded=0, speed_in_mm_per_min=3000.0, acceleration_in_mm_per_s2=50.0, teachColor=BLUE, combo1=MachineMotion1, combo2=(1) Custom Actuator, combo3=Home, combo6=In series, message=Homing, description=Moves the actuator in the negative direction until the home sensor is triggered and sets position to zero (0)., comboAddress=Address 1, comboActuator=Valve 1)
      Script: extrude_knife3()
      URCap MachineLogic for Universal Robots (MachineLogic for Universal Robots, Vention Inc.) dataModel(type=addMotor, numberAdded=0, speed_in_mm_per_min=3000.0, acceleration_in_mm_per_s2=50.0, ActuatorPos=lch, teachColor=BLUE, combo1=MachineMotion1, combo2=(1) Custom Actuator, combo3=Move to Position, combo6=In series, message=Move to Position, description=Moves the actuator to a specified position from the home location., comboAddress=Address 1, comboActuator=Valve 1)
    Else 
      Script: extrude_knife3()
  SuppressedNode
    Script: move_path_cover_left3()
  SuppressedNode
    pointtopvcham := pathturn[0]
  SuppressedNode
    URCap MachineLogic for Universal Robots (MachineLogic for Universal Robots, Vention Inc.) dataModel(type=addMotor, numberAdded=0, speed_in_mm_per_min=3000.0, acceleration_in_mm_per_s2=50.0, ActuatorPos=liftcolumnzneeded, teachColor=BLUE, combo1=MachineMotion1, combo2=(1) Custom Actuator, combo3=Move to Position, combo6=In series, message=Move to Position, description=Moves the actuator to a specified position from the home location., comboAddress=Address 1, comboActuator=Valve 1)
  SuppressedNode
    MoveJ speed 60 deg/s, acceleration 80 deg/s^2 (useActiveTCP=true optimoveEnabled=false optiMoveSpeed=0.3 optiMoveAcceleration=0.09) feature=Base
      Waypoint Variable (Variable): variable=pointtopvcham
  Script: align_for_cover_straight()
  Script: move_path_cover_lt()
  MoveJ speed 60 deg/s, acceleration 80 deg/s^2 (useActiveTCP=true optimoveEnabled=false optiMoveSpeed=0.3 optiMoveAcceleration=0.09) feature=Base
    Waypoint Waypoint_8: TCP in base x=-262.599 y=-117.911 z=443.767 mm, rx=0.1153 ry=3.1146 rz=0.2657 rad; joints [5.497, -142.032, 129.309, 13.11, 99.793, -9.621] deg; TCP offset x=-9.5 y=-328 z=105.73 mm, rx=1.2092 ry=-1.2092 rz=1.2092 rad
    Waypoint Waypoint_9: TCP in base x=397.354 y=356.263 z=319.809 mm, rx=2.3163 ry=2.0576 rz=0.0741 rad; joints [-198.308, -118.162, 133.452, -12.561, -11.517, -6.326] deg
  URCap MachineLogic for Universal Robots (MachineLogic for Universal Robots, Vention Inc.) dataModel(type=addMotor, numberAdded=0, speed_in_mm_per_min=3000.0, acceleration_in_mm_per_s2=50.0, teachColor=BLUE, combo1=MachineMotion1, combo2=(1) Custom Actuator, combo3=Home, combo6=In series, message=Homing, description=Moves the actuator in the negative direction until the home sensor is triggered and sets position to zero (0)., comboAddress=Address 1, comboActuator=Valve 1)
  SafeHome (positionOptionType=SPEED_AND_ACCELERATION speed=1.047198 acceleration=1.396263 nextMotionTime=2)
SubProgram Test_Teach_Cover_LT (keepSynchronizedWithDisk=false) programFile=/programs/Test Teach Cover LT.urp
  Set NoAction tcp=pretend_w_top
  SuppressedNode
    MoveL speed 250 mm/s, acceleration 1200 mm/s^2 (useActiveTCP=true optimoveEnabled=false optiMoveSpeed=0.3 optiMoveAcceleration=0.09) feature=Base
      Waypoint Waypoint_1: TCP in base x=183.613 y=373.491 z=464.002 mm, rx=0 ry=3.1416 rz=0 rad; joints [-144.817, -120.486, 148.461, -117.931, -90.033, 125.101] deg; TCP offset x=0 y=0 z=19 mm, rx=0 ry=0 rz=0 rad
      'move welder up out of holder'
  MoveJ speed 60 deg/s, acceleration 80 deg/s^2 (useActiveTCP=false optimoveEnabled=false optiMoveSpeed=0.3 optiMoveAcceleration=0.09) tcp=TCP_1_plate; feature=Base
    Waypoint Waypoint_40: TCP in base x=360.688 y=270.12 z=646.145 mm, rx=0.0578 ry=2.126 rz=2.1341 rad; joints [-198.126, -117.852, 133.303, -13.01, -11.422, -6.036] deg
    'above waypoint is home'
    SuppressedNode
      Waypoint Waypoint_2: TCP in base x=-548.957 y=386.285 z=143.71 mm, rx=1.5708 ry=0 rz=0 rad; joints [-60.253, -57.926, 123.544, -65.529, -60.311, -0.099] deg
    Waypoint Waypoint_1: TCP in base x=-565.561 y=-88.282 z=748.934 mm, rx=0.347 ry=3.1015 rz=-0.0385 rad; joints [-12.028, -113.359, 121.362, 263.351, -88.693, -89.284] deg
  Set NoAction tcp=pretend_w_top
  freedrive_m_var := False
  freedrive_m_var := True
  Popup Message (haltProgram=false message=Move the TCP to the left side of the weld (very center of groove), then click 'Continue' inputType=Text)
  tcp_pose_left := get_actual_tcp_pose()
  Popup Message (haltProgram=false message=Move the TCP to the right side of the weld (very center of groove), then click 'Continue' inputType=Text)
  tcp_pose_right := get_actual_tcp_pose()
  freedrive_m_var := False
  Wait Sleep waitTime=0.25
  Script: sync()
SubProgram move_path_cover_lt (keepSynchronizedWithDisk=false) programFile=/programs/move_path_cover_lt.urp
  p1 := pathturn[0]
  p2 := pathturn[1]
  p3 := pathturn[2]
  p4 := pathturn[3]
  p5 := pathturn[4]
  p6 := pathturn[5]
  pa1 := p[p1[0],p1[1],p1[2]+0.05,p1[3],p1[4],p1[5]]
  pret := p[p6[0],p6[1],p6[2]+0.05,p6[3],p6[4],p6[5]]
  'go to preheat'
  Set NoAction tcp=pretend_welder
  If 1≟2
    'testing bs'
    Set NoAction tcp=pretend_w_top
  MoveJ speed 60 deg/s, acceleration 80 deg/s^2 (useActiveTCP=true optimoveEnabled=false optiMoveSpeed=0.3 optiMoveAcceleration=0.09) feature=Base
    Waypoint Variable (Variable): variable=pa1
  MoveL speed 50 mm/s, acceleration 50 mm/s^2 (useActiveTCP=true optimoveEnabled=false optiMoveSpeed=0.3 optiMoveAcceleration=0.09) feature=Base
    Waypoint Variable (Variable): variable=p1
  Wait Sleep waitTime=4
  URCap WireTank Serial (WireTank Serial, WireTank, LLC) dataModel(NODE_TITLE=Serial Bridge uR1, Command=[252,82,49], QUERY=false, OUTPUT_ENTRY=Static, byte_array=true, Variable(key=OUTPUT_VARIABLE, variable=HwResp))
  Set DigitalOutput pin=digital_out[0]; digitalValue=1
  Wait Sleep waitTime=1
  MoveL speed 9 mm/s, acceleration 1200 mm/s^2 (useActiveTCP=true optimoveEnabled=false optiMoveSpeed=0.3 optiMoveAcceleration=0.09) feature=Base
    Waypoint Variable (Variable): variable=p2
    Waypoint Variable (Variable): variable=p3
    Waypoint Variable (Variable): variable=p4
    Waypoint Variable (Variable): variable=p5
  SuppressedNode
    If deepcham removedSiblings(If(type=Else checkContinuously=false, children(Move(motionType=MoveL speed=0.01 acceleration=1.2 useActiveTCP=true positionType=CartesianPose optimoveEnabled=false optiMoveSpeed=0.3 optiMoveAcceleration=0.09, feature=Base, children(Waypoint(type=Variable name=Variable, variable=p2), Waypoint(type=Variable name=Variable, variable=p3), Waypoint(type=Variable name=Variable, variable=p4), Waypoint(type=Variable name=Variable, variable=p5))))))
      MoveL speed 7 mm/s, acceleration 1200 mm/s^2 (useActiveTCP=true optimoveEnabled=false optiMoveSpeed=0.3 optiMoveAcceleration=0.09) feature=Base
        Waypoint Variable (Variable): variable=p2
        Waypoint Variable (Variable): variable=p3
        Waypoint Variable (Variable): variable=p4
        Waypoint Variable (Variable): variable=p5
  URCap WireTank Serial (WireTank Serial, WireTank, LLC) dataModel(QUERY=false, NODE_TITLE=Serial Bridge uR0, Command=[252,82,48], OUTPUT_ENTRY=Static, byte_array=true, Variable(key=OUTPUT_VARIABLE, variable(name=HwResp)))
  Set DigitalOutput pin=digital_out[0]; digitalValue=0
  MoveL speed 10 mm/s, acceleration 1200 mm/s^2 (useActiveTCP=true optimoveEnabled=false optiMoveSpeed=0.3 optiMoveAcceleration=0.09) feature=Base
    Waypoint Variable (Variable): variable=p6
  Wait Sleep waitTime=1
  MoveL speed 50 mm/s, acceleration 50 mm/s^2 (useActiveTCP=true optimoveEnabled=false optiMoveSpeed=0.3 optiMoveAcceleration=0.09) feature=Base
    Waypoint Variable (Variable): variable=pret
SubProgram align_for_cover_straight (keepSynchronizedWithDisk=false) programFile=/programs/align for cover straight.urp
  SuppressedNode
    Folder dummypoints
      MoveJ speed 60 deg/s, acceleration 80 deg/s^2 (useActiveTCP=true optimoveEnabled=false optiMoveSpeed=0.3 optiMoveAcceleration=0.09) feature=Base
        Waypoint oldhome: TCP in base x=397.354 y=356.263 z=319.809 mm, rx=2.3163 ry=2.0576 rz=0.0741 rad; joints [-198.308, -118.162, 133.452, -12.561, -11.517, -6.326] deg; TCP offset x=-9.5 y=-328 z=105.73 mm, rx=1.2092 ry=-1.2092 rz=1.2092 rad
        Waypoint demo: TCP in base x=-1245.427 y=-117.911 z=443.767 mm, rx=0.1153 ry=3.1146 rz=0.2657 rad; joints [0.095, -71.189, 81.089, -9.527, 94.427, -9.693] deg
        Waypoint Waypoint_1: TCP in base x=-262.599 y=-117.911 z=443.767 mm, rx=0.1153 ry=3.1146 rz=0.2657 rad; joints [5.497, -142.032, 129.309, 13.11, 99.793, -9.621] deg
  MoveJ speed 60 deg/s, acceleration 80 deg/s^2 (useActiveTCP=true optimoveEnabled=false optiMoveSpeed=0.3 optiMoveAcceleration=0.09) feature=Base
    Waypoint Waypoint_6: TCP in base x=397.354 y=356.263 z=319.809 mm, rx=2.3163 ry=2.0576 rz=0.0741 rad; joints [-198.308, -118.162, 133.452, -12.561, -11.517, -6.326] deg
    Waypoint Waypoint_5: TCP in base x=-169.948 y=714.519 z=357.695 mm, rx=1.393 ry=2.6763 rz=-0.2105 rad; joints [-106.374, -98.913, 115.606, -1.537, 39.342, -7.787] deg; TCP offset x=-11.7 y=-328 z=105 mm, rx=1.2092 ry=-1.2092 rz=1.2092 rad
    Waypoint Waypoint_7: TCP in base x=-262.599 y=-117.911 z=443.767 mm, rx=0.1153 ry=3.1146 rz=0.2657 rad; joints [5.497, -142.032, 129.309, 13.11, 99.793, -9.621] deg; TCP offset x=-9.5 y=-328 z=105.73 mm, rx=1.2092 ry=-1.2092 rz=1.2092 rad
  If 1≟1
    If is_xvcut(pathturn[1],pathturn[2])
      MoveJ speed 60 deg/s, acceleration 80 deg/s^2 (useActiveTCP=true optimoveEnabled=false optiMoveSpeed=0.3 optiMoveAcceleration=0.09) feature=Base
        Waypoint Waypoint_4: TCP in base x=-433.665 y=-217.871 z=358.002 mm, rx=-1.8955 ry=2.499 rz=0.0369 rad; joints [-38.305, -120.231, 130.629, -13.018, -22.753, 1.506] deg; TCP offset x=-9.27 y=-328 z=105.71 mm, rx=1.2092 ry=-1.2092 rz=1.2092 rad
        'this is for xvcut'
SubProgram extrude_knife3 (keepSynchronizedWithDisk=false) programFile=/programs/extrude_knife3.urp
  Folder pre program stuff
    Set NoAction tcp=pretend_welder
    ek_sp := get_actual_tcp_pose()
    MoveL speed 5 mm/s, acceleration 1200 mm/s^2 (useActiveTCP=true optimoveEnabled=false optiMoveSpeed=0.3 optiMoveAcceleration=0.09) feature=Base
      Waypoint Variable (Variable): variable=ek_sp
  'list possible points'
  Folder robot 1 moves
    If 1≟2
      MoveJ speed 60 deg/s, acceleration 80 deg/s^2 (useActiveTCP=true optimoveEnabled=false optiMoveSpeed=0.3 optiMoveAcceleration=0.09) feature=Base
        Waypoint r1_ek_oldhome: TCP in base x=397.38 y=356.254 z=319.821 mm, rx=2.3163 ry=2.0576 rz=0.0741 rad; joints [-198.126, -117.851, 133.303, -13.009, -11.422, -6.035] deg; TCP offset x=-5.49 y=-328 z=106.39 mm, rx=1.2092 ry=-1.2092 rz=1.2092 rad
        Waypoint r1_ek_extrude: TCP in base x=454.852 y=405.449 z=64.015 mm, rx=2.3168 ry=2.0514 rz=0.0767 rad; joints [-187.624, -89.406, 141.395, -19.732, -0.818, -36.116] deg
        Waypoint r1_ek_front: TCP in base x=439.065 y=405.452 z=65.996 mm, rx=2.3168 ry=2.0514 rz=0.0766 rad; joints [-187.962, -93.321, 143.386, -27.168, -1.131, -26.752] deg
        Waypoint r1_ek_middle: TCP in base x=419.01 y=404.851 z=65.995 mm, rx=2.3096 ry=2.0447 rz=0.0891 rad; joints [-188.553, -97.485, 146.002, -33.769, -1.69, -19.324] deg
        Waypoint r1_ek_middle2: TCP in base x=417.012 y=405.435 z=65.003 mm, rx=2.3169 ry=2.0513 rz=0.0766 rad; joints [-188.493, -97.025, 145.794, -33.21, -1.638, -19.415] deg
        Waypoint r1_ek_bottom: TCP in base x=413.072 y=405.431 z=68 mm, rx=2.3168 ry=2.0513 rz=0.0767 rad; joints [-188.596, -97.887, 146.02, -33.517, -1.738, -18.475] deg
        Waypoint r1_ek_end: TCP in base x=389.999 y=405.444 z=68.005 mm, rx=2.3169 ry=2.0514 rz=0.0766 rad; joints [-189.248, -101.07, 148.002, -36.337, -2.38, -14.447] deg
  Folder robot 2 moves
    If 1≟2
      MoveJ speed 60 deg/s, acceleration 80 deg/s^2 (useActiveTCP=true optimoveEnabled=false optiMoveSpeed=0.3 optiMoveAcceleration=0.09) feature=Base
        Waypoint r2_ek_oldhome: TCP in base x=397.38 y=356.254 z=319.821 mm, rx=2.3163 ry=2.0576 rz=0.0741 rad; joints [-198.308, -118.162, 133.451, -12.562, -11.515, -6.325] deg; TCP offset x=-9.5 y=-328 z=105.73 mm, rx=1.2092 ry=-1.2092 rz=1.2092 rad
        SuppressedNode
          Waypoint Waypoint_1: TCP in base x=612.886 y=429.305 z=100.477 mm, rx=1.8619 ry=2.4807 rz=0.0957 rad; joints [-182.793, -81.736, 125.569, -42.478, -18.966, -5.44] deg
        Waypoint r2_ek_extrude: TCP in base x=612.886 y=429.305 z=100.477 mm, rx=2.15 ry=2.2258 rz=0.0874 rad; joints [-183.316, -85.158, 129.692, -39.696, -5.262, -8.969] deg
        Waypoint r2_ek_front: TCP in base x=556.405 y=429.305 z=76.984 mm, rx=-2.1704 ry=-2.2682 rz=-0.0159 rad; joints [-183.513, -85.623, 132.794, -41.666, -5.994, -5.809] deg
        Waypoint r2_ek_middle: TCP in base x=550.034 y=429.305 z=76.254 mm, rx=-2.1704 ry=-2.2682 rz=-0.0159 rad; joints [-183.554, -85.983, 133.283, -41.831, -6.035, -5.773] deg
        Waypoint r2_ek_bottom: TCP in base x=546.595 y=429.305 z=80.868 mm, rx=-2.1704 ry=-2.2682 rz=-0.0159 rad; joints [-183.576, -86.513, 133.34, -41.373, -6.058, -5.758] deg
        Waypoint r2_ek_end: TCP in base x=537.335 y=429.305 z=80.868 mm, rx=-2.1704 ry=-2.2682 rz=-0.0159 rad; joints [-183.639, -87.118, 134.001, -41.482, -6.12, -5.705] deg
  Folder robot 3 moves
    If 1≟2
      MoveJ speed 60 deg/s, acceleration 80 deg/s^2 (useActiveTCP=true optimoveEnabled=false optiMoveSpeed=0.3 optiMoveAcceleration=0.09) feature=Base
        Waypoint r3_ek_oldhome: TCP in base x=397.386 y=356.252 z=369.81 mm, rx=2.3163 ry=2.0576 rz=0.0741 rad; joints [-198.244, -119.435, 129.987, -8.275, -11.561, -5.872] deg; TCP offset x=-11.7 y=-328 z=105 mm, rx=1.2092 ry=-1.2092 rz=1.2092 rad
        Waypoint r3_ek_extrude: TCP in base x=612.884 y=429.31 z=150 mm, rx=2.15 ry=2.2258 rz=0.0874 rad; joints [-183.233, -88.144, 127.755, -35.039, -5.316, -8.705] deg
        Waypoint r3_ek_front: TCP in base x=585.402 y=429.31 z=130.897 mm, rx=-2.1411 ry=-2.2788 rz=0.0035 rad; joints [-183.22, -86.46, 127.828, -36.419, -6.878, -4.248] deg; TCP offset x=-9.27 y=-328 z=105.71 mm, rx=1.2092 ry=-1.2092 rz=1.2092 rad
        Waypoint r3_ek_middle: TCP in base x=557.524 y=429.31 z=129.294 mm, rx=-2.1411 ry=-2.2788 rz=0.0035 rad; joints [-183.379, -88.209, 129.87, -36.837, -7.04, -4.124] deg
        Waypoint r3_ek_bottom: TCP in base x=555.664 y=429.31 z=134.686 mm, rx=-2.1411 ry=-2.2788 rz=0.0035 rad; joints [-183.391, -88.643, 129.758, -36.302, -7.051, -4.111] deg
        Waypoint r3_ek_end: TCP in base x=526.089 y=429.31 z=134.686 mm, rx=-2.1411 ry=-2.2788 rz=0.0035 rad; joints [-183.58, -90.668, 131.798, -36.459, -7.243, -3.97] deg
  Folder robot 4 moves
    If 1≟2
      MoveJ speed 60 deg/s, acceleration 80 deg/s^2 (useActiveTCP=true optimoveEnabled=false optiMoveSpeed=0.3 optiMoveAcceleration=0.09) feature=Base
        Waypoint r4_ek_oldhome: TCP in base x=397.38 y=356.254 z=319.821 mm, rx=2.3163 ry=2.0576 rz=0.0741 rad; joints [-198.707, -118.624, 133.667, -13.08, -11.814, -5.554] deg; TCP offset x=-11.7 y=-328 z=105 mm, rx=1.2092 ry=-1.2092 rz=1.2092 rad
        Waypoint r4_ek_extrude: TCP in base x=458.671 y=429.305 z=125.141 mm, rx=2.15 ry=2.2258 rz=0.0874 rad; joints [-184.739, -98.178, 139.464, -38.783, -6.613, -6.625] deg
        Waypoint r4_ek_front: TCP in base x=420.084 y=429.305 z=122.37 mm, rx=-2.2067 ry=-2.1774 rz=0.0527 rad; joints [-184.629, -98.923, 139.999, -38.069, -3.732, -0.951] deg; TCP offset x=-6.9 y=-329 z=104.9 mm, rx=1.222 ry=-1.2009 rz=1.222 rad
        Waypoint r4_ek_middle: TCP in base x=385.664 y=429.305 z=119.862 mm, rx=-2.2067 ry=-2.1774 rz=0.0527 rad; joints [-185.039, -101.657, 142.224, -37.721, -4.144, -0.789] deg
        Waypoint r4_ek_bottom: TCP in base x=385.664 y=429.305 z=122.81 mm, rx=-2.2067 ry=-2.1774 rz=0.0527 rad; joints [-185.04, -101.863, 142.06, -37.349, -4.144, -0.791] deg
        Waypoint r4_ek_end: TCP in base x=366.757 y=429.305 z=122.81 mm, rx=-2.2067 ry=-2.1774 rz=0.0527 rad; joints [-185.301, -103.548, 143.17, -36.87, -4.406, -0.695] deg
  'detemine correct points for which robot'
  If robot_number≟1
    Folder robot1 positions
      ek_oldhome := r1_ek_oldhome_p
      ek_extrude := r1_ek_extrude_p
      ek_front := r1_ek_front_p
      ek_middle := r1_ek_middle_p
      ek_middle2 := r1_ek_middle2_p
      ek_bottom := r1_ek_bottom_p
      ek_end := r1_ek_end_q
  ElseIf robot_number≟2
    Folder robot2 positions
      ek_oldhome := r2_ek_oldhome_p
      ek_extrude := r2_ek_extrude_p
      ek_front := r2_ek_front_p
      ek_middle := r2_ek_middle_p
      ek_middle2 := r2_ek_middle_p
      ek_bottom := r2_ek_bottom_p
      ek_end := r2_ek_end_q
  ElseIf robot_number≟3
    Folder robot3 positions
      ek_oldhome := r3_ek_oldhome_p
      ek_extrude := r3_ek_extrude_p
      ek_front := r3_ek_front_p
      ek_middle := r3_ek_middle_p
      ek_middle2 := r3_ek_middle_p
      ek_bottom := r3_ek_bottom_p
      ek_end := r3_ek_end_q
  ElseIf robot_number≟4
    Folder robot4 positions
      ek_oldhome := r4_ek_oldhome_p
      ek_extrude := r4_ek_extrude_p
      ek_front := r4_ek_front_p
      ek_middle := r4_ek_middle_p
      ek_middle2 := r4_ek_middle_p
      ek_bottom := r4_ek_bottom_p
      ek_end := r4_ek_end_q
  'start of program'
  SuppressedNode
    SafeHome (positionOptionType=SPEED_AND_ACCELERATION speed=1.047198 acceleration=1.396263 nextMotionTime=2)
  Set NoAction tcp=pretend_welder
  MoveJ speed 60 deg/s, acceleration 80 deg/s^2 (useActiveTCP=true positionType=JointAngles optimoveEnabled=false optiMoveSpeed=0.3 optiMoveAcceleration=0.09) feature=Base
    Waypoint Waypoint_3: TCP in base x=397.386 y=356.252 z=369.81 mm, rx=2.3163 ry=2.0576 rz=0.0741 rad; joints [-198.287, -119.237, 129.894, -8.387, -11.604, -5.865] deg; TCP offset x=-9.27 y=-328 z=105.71 mm, rx=1.2092 ry=-1.2092 rz=1.2092 rad
    'joint angles for fixed position'
  MoveJ speed 60 deg/s, acceleration 80 deg/s^2 (useActiveTCP=true optimoveEnabled=false optiMoveSpeed=0.3 optiMoveAcceleration=0.09) feature=Base
    SuppressedNode
      Waypoint r1_ek_oldhome: TCP in base x=397.38 y=356.254 z=319.821 mm, rx=2.3163 ry=2.0576 rz=0.0741 rad; joints [-198.126, -117.851, 133.303, -13.009, -11.422, -6.035] deg; TCP offset x=-5.49 y=-328 z=106.39 mm, rx=1.2092 ry=-1.2092 rz=1.2092 rad
    Waypoint Variable (Variable): variable=ek_oldhome
    'above waypoint is home'
  'move above bucket'
  MoveJ speed 60 deg/s, acceleration 80 deg/s^2 (useActiveTCP=true optimoveEnabled=false optiMoveSpeed=0.3 optiMoveAcceleration=0.09) feature=Base
    SuppressedNode
      Waypoint r1_ek_extrude: TCP in base x=454.852 y=405.449 z=64.015 mm, rx=2.3168 ry=2.0514 rz=0.0767 rad; joints [-187.624, -89.406, 141.395, -19.732, -0.818, -36.116] deg
    Waypoint Variable (Variable): variable=ek_extrude
  'extrude out a foot'
  SuppressedNode
    Script: turn_extrusion_on()
  URCap WireTank Serial (WireTank Serial, WireTank, LLC) dataModel(NODE_TITLE=Serial Bridge uR1, Command=[252,82,49], QUERY=false, byte_array=true, OUTPUT_ENTRY=Static, Variable(key=OUTPUT_VARIABLE, variable(name=HwResp)))
  Set DigitalOutput pin=digital_out[0]; digitalValue=1
  Wait Sleep waitTime=4
  URCap WireTank Serial (WireTank Serial, WireTank, LLC) dataModel(QUERY=false, NODE_TITLE=Serial Bridge uR0, Command=[252,82,48], byte_array=true, OUTPUT_ENTRY=Static, Variable(key=OUTPUT_VARIABLE, variable=HwResp))
  Wait Sleep waitTime=1
  Set DigitalOutput pin=digital_out[0]; digitalValue=0
  'slice'
  MoveL speed 30 mm/s, acceleration 50 mm/s^2 (useActiveTCP=true optimoveEnabled=false optiMoveSpeed=0.3 optiMoveAcceleration=0.09) feature=Base
    SuppressedNode
      Waypoint r1_ek_front: TCP in base x=439.065 y=405.452 z=65.996 mm, rx=2.3168 ry=2.0514 rz=0.0766 rad; joints [-187.962, -93.321, 143.386, -27.168, -1.131, -26.752] deg
    SuppressedNode
      Waypoint r1_ek_middle: TCP in base x=419.01 y=404.851 z=65.995 mm, rx=2.3096 ry=2.0447 rz=0.0891 rad; joints [-188.553, -97.485, 146.002, -33.769, -1.69, -19.324] deg
    SuppressedNode
      Waypoint r1_ek_middle2: TCP in base x=417.012 y=405.435 z=65.003 mm, rx=2.3169 ry=2.0513 rz=0.0766 rad; joints [-188.493, -97.025, 145.794, -33.21, -1.638, -19.415] deg
    SuppressedNode
      Waypoint r1_ek_bottom: TCP in base x=413.072 y=405.431 z=68 mm, rx=2.3168 ry=2.0513 rz=0.0767 rad; joints [-188.596, -97.887, 146.02, -33.517, -1.738, -18.475] deg
    SuppressedNode
      Waypoint r1_ek_end: TCP in base x=389.999 y=405.444 z=68.005 mm, rx=2.3169 ry=2.0514 rz=0.0766 rad; joints [-189.248, -101.07, 148.002, -36.337, -2.38, -14.447] deg
    Waypoint Variable (Variable): variable=ek_front
    Waypoint Variable (Variable): variable=ek_middle
    Waypoint Variable (Variable): variable=ek_middle2
    Waypoint Variable (Variable): variable=ek_bottom
    Waypoint Variable (Variable): variable=ek_end
  MoveJ speed 60 deg/s, acceleration 80 deg/s^2 (useActiveTCP=true optimoveEnabled=false optiMoveSpeed=0.3 optiMoveAcceleration=0.09) feature=Base
    SuppressedNode
      Waypoint r1_ek_oldhome: TCP in base x=397.38 y=356.254 z=319.821 mm, rx=2.3163 ry=2.0576 rz=0.0741 rad; joints [-198.126, -117.851, 133.303, -13.009, -11.422, -6.035] deg
    Waypoint Variable (Variable): variable=ek_oldhome
    'above waypoint is home'
  SuppressedNode
    SafeHome (positionOptionType=SPEED_AND_ACCELERATION speed=1.047198 acceleration=1.396263 nextMotionTime=2)
SubProgram Cover_LT_Homing (keepSynchronizedWithDisk=false) programFile=/programs/Cover LT Homing.urp
  Set NoAction tcp=pretend_w_top
  'assume the person has just taught the right point and pressed continue.'
  SuppressedNode
    SafeHome (positionOptionType=SPEED_AND_ACCELERATION speed=1.047198 acceleration=1.396263 nextMotionTime=2)
  SuppressedNode
    MoveJ speed 60 deg/s, acceleration 80 deg/s^2 (useActiveTCP=true optimoveEnabled=false optiMoveSpeed=0.3 optiMoveAcceleration=0.09) feature=Base
      Waypoint demo_point0: TCP in base x=-1268.829 y=243.799 z=397.866 mm, rx=1.3918 ry=-0.5735 rz=-1.0174 rad; joints [-39.169, -62.377, 106.188, -68.476, 20.677, 9.969] deg; TCP offset x=-1.032 y=-18.062 z=285.234 mm, rx=0 ry=0 rz=0 rad
  SuppressedNode
    MoveJ speed 60 deg/s, acceleration 80 deg/s^2 (useActiveTCP=true optimoveEnabled=false optiMoveSpeed=0.3 optiMoveAcceleration=0.09) feature=Base
      Waypoint Waypoint_1: TCP in base x=-726.76 y=313.857 z=-3.219 mm, rx=-0.1302 ry=-1.6605 rz=-0.1403 rad; joints [-65.067, -50.619, 153.092, -93.35, 35.027, 81.724] deg; TCP offset x=0 y=0 z=246 mm, rx=0 ry=0 rz=0 rad
      Waypoint Waypoint_2: TCP in base x=-1013.668 y=283.774 z=13.404 mm, rx=-0.1302 ry=-1.6605 rz=-0.1403 rad; joints [-36.803, -53.188, 133.142, -74.065, 63.057, 86.565] deg
  Wait Sleep waitTime=1
  SuppressedNode
    tp := get_actual_tcp_pose()
  SuppressedNode
    Script file /programs/analyze_touchpoints.script
      | # this file creates the function for analyzing touchpoints
      | # define pi
      | pi = 3.1415926535
      | # initialize a lift column extension needed of 0.0
      | global liftcolumnzneeded = 0.0 # set this variable in mm
      | 
      | # this is the main entry point for calculations.
      | # it takes in the 5 points, analyzes the shape of the box, and then calculates path points and returns them
      | # specifically for Down, Over, then Around (DOtA)
      | # specifically for right-sided boxes (vertical weld on right side of edge)
      | def main_calculate_right(p11, p12, p21, p22, p3, p13, p23, chamferover):
      |     struct1 = analyze_touchpoints_only(p11, p12, p21, p22, p3)
      |     list1 = analyze_vertical_touchpoints(p11, p12, p13, p21, p22, p23, p3)
      |     struct2 = calculate_DOtA_points_right(struct1, list1, chamferover)
      |     validity = check_validity_right(struct1, struct2)
      |     return struct2
      | end
      | 
      | # this is the main entry point for calculations.
      | # it takes in the 5 points, analyzes the shape of the box, and then calculates path points and returns them
      | # specifically for Down, Over, then Around (DOtA)
      | # specifically for left-sided boxes (vertical weld on left side of edge)
      | def main_calculate_left(p11, p12, p21, p22, p3, p13, p23, chamferover):
      |     struct1 = analyze_touchpoints_only(p11, p12, p21, p22, p3)
      |     list1 = analyze_vertical_touchpoints(p11, p12, p13, p21, p22, p23, p3)
      |     struct2 = calculate_DOtA_points_left(struct1, list1, chamferover)
      |     validity = check_validity_left(struct1, struct2)
      |     return struct2
      | end
      | 
      | # this is the main entry point for calculations, for Floor Corner Extended.
      | # it takes in the 7 touchpoints, analyzes the shape of the box.
      | # takes in the user defined point for the top of the weld (tcp_pose_top) and then calculates path points
      | # loopingly tries to calculate the extension along the sidewall that fulfills get_inverse_kin_has_solution() and provides the farthest extension possible
      | # returns the pathpoints
      | # specifically for Down, Over, then Around (DOtA)
      | # specifically for right-sided boxes (vertical weld on right side of edge)
      | def main_calculate_right_extended(p11, p12, p21, p22, p3, p13, p23, chamferover, chamferup, tcp_pose_top):
      |     struct1 = analyze_touchpoints_only(p11, p12, p21, p22, p3)
      |     list1 = analyze_vertical_touchpoints(p11, p12, p13, p21, p22, p23, p3)
      |     struct2 = calculate_DOtA_points_right_extended(struct1, list1, chamferover, chamferup, tcp_pose_top)
      |     struct3 = check_validity_right(struct1, struct2)
      |     return struct3
      | end
      | 
      | # this is the main entry point for calculations, for Floor Corner Extended.
      | # it takes in the 7 touchpoints, analyzes the shape of the box.
      | # takes in the user defined point for the top of the weld (tcp_pose_top) and then calculates path points
      | # loopingly tries to calculate the extension along the sidewall that fulfills get_inverse_kin_has_solution() and provides the farthest extension possible
      | # returns the pathpoints
      | # specifically for Down, Over, then Around (DOtA)
      | # specifically for left-sided boxes (vertical weld on left side of edge)
      | def main_calculate_left_extended(p11, p12, p21, p22, p3, p13, p23, chamferover, chamferup, tcp_pose_top):
      |     struct1 = analyze_touchpoints_only(p11, p12, p21, p22, p3)
      |     list1 = analyze_vertical_touchpoints(p11, p12, p13, p21, p22, p23, p3)
      |     struct2 = calculate_DOtA_points_left_extended(struct1, list1, chamferover, chamferup, tcp_pose_top)
      |     struct3 = check_validity_left(struct1, struct2)
      |     return struct3
      | end
      | 
      | # it takes 5 arguments as points
      | # it returns a struct containing: (pointintersect, pointapproach1, pointapproach2, point1, point2, point3, point4, point5, pointreturn1, heading1, heading2, heading3, path2r1, path2r2, path2l1, path2l2)
      | # specifically for Around then Up (AtU)
      | def analyze_touchpoints(p11, p12, p21, p22, p3):
      |   # FIND THE INTERSECTION
      |   # comment get the z
      |   zcoord=p3[2]
      | 
      |   # get the raw points from the first line
      |   l1p1x=p11[0]
      |   l1p1y=p11[1]
      |   l1p2x=p12[0]
      |   l1p2y=p12[1]
      | 
      |   # equate the first line in 2d space
      |   ml1 = (l1p2y-l1p1y) / (l1p2x-l1p1x)
      | 
      |   # b = y - mx
      |   bl1 = l1p1y - ml1 * l1p1x
      | 
      |   # get the raw points from the second line
      |   l2p1x=p21[0]
      |   l2p1y=p21[1]
      |   l2p2x=p22[0]
      |   l2p2y=p22[1]
      | 
      |   # equate the second line in 2d space
      |   ml2 = (l2p2y-l2p1y) / (l2p2x-l2p1x)
      | 
      |   # b = y - mx
      |   bl2 = l2p1y - ml2 * l2p1x
      | 
      | 
      |   # find the intersection of the two lines
      |   # m1x+b1 = m2x+b2
      |   # m1x - m2x = b2 - b1
      |   # x = (b2-b1) / (m1-m2)
      |   xintersect = (bl2-bl1) / (ml1-ml2)
      |   yintersect = ml1 * xintersect + bl1
      | 
      |   #FIND THE VECTORS
      |   #define a vector from the intersection to the second point on the first line
      |   l1delxfull = l1p2x - xintersect
      |   l1delyfull = l1p2y - yintersect
      | 
      |   l1delmag = sqrt(l1delxfull*l1delxfull + l1delyfull*l1delyfull)
      | 
      |   l1delxunit = l1delxfull / l1delmag
      |   l1delyunit = l1delyfull / l1delmag
      | 
      |   #define a vector from the intersection to the second point on the second line
      |   l2delxfull = l2p2x - xintersect
      |   l2delyfull = l2p2y - yintersect
      | 
      |   l2delmag = sqrt(l2delxfull*l2delxfull + l2delyfull*l2delyfull)
      | 
      |   l2delxunit = l2delxfull / l2delmag
      |   l2delyunit = l2delyfull / l2delmag
      | 
      |   # FIND THE FOUR POINTS ON THE LINES
      |   # find locations 8 inches away from  intersect point
      |   # CONST
      |   welddistance = 8
      |   roundoverdistance = 0.05
      |   zup = .375
      |   # inches
      |   wd = welddistance * 25.4 / 1000
      |   rod = roundoverdistance * 25.4 / 1000
      |   zup = zup * 25.4 / 1000
      | 
      |   # now we have the unit vector. extend the weld distance from the intersection
      |   x = xintersect + l1delxunit * wd
      |   y = yintersect + l1delyunit * wd
      |   z = zcoord + zup
      | 
      |   point1 = p[x,y,z,1.570796,0,0] # dummy orientation for now
      | 
      |   x = xintersect + l1delxunit * rod
      |   y = yintersect + l1delyunit * rod
      | 
      |   point2 = p[x,y,z,1.570796,0,0]
      | 
      |   # now we have the unit vector. extend the weld distance from the intersection
      |   x = xintersect + l2delxunit * wd
      |   y = yintersect + l2delyunit * wd
      | 
      |   point5 = p[x,y,z,0,-1.570796,0]
      | 
      |   x = xintersect + l2delxunit * rod
      |   y = yintersect + l2delyunit * rod
      | 
      |   point4 = p[x,y,z,0,-1.570796,0]
      | 
      |   #DEFINE APPROACH POINTS
      |   pointintersect = p[xintersect,yintersect,zcoord,0,0,0]
      |   pointapproach1 = p[xintersect+0.1,yintersect+0.1,z,1.570796,0,0]
      |   pointapproach2 = p[point1[0], point1[1]+0.1, point1[2], point1[3], point1[4], point1[5]]
      |   pointreturn1 = p[point5[0]+0.1, point5[1], point5[2], point5[3], point5[4], point5[5]]
      | 
      |   #FIND HEADINGS
      |   #for each heading, find the angle of the line with respect to the pos x axis. then add/subtract 90 degrees because you want to be perpendicular to that
      |   headingvector1 = convert_uv_to_heading(l1delxunit, l1delyunit)
      |   headingvector2 = convert_uv_to_heading(l2delxunit, l2delyunit)
      |   # find halfway heading
      |   heading2 = (headingvector1 + headingvector2)/2
      |   # find headings that the robot should face while traveling, perpendicular to the vectors of the sides of the box
      |   heading1 = headingvector1 + pi/2
      |   heading3 = headingvector2 - pi/2
      | 
      |   #FIND POINT 3
      |   #see if we have to / can find point 3
      |   findpoint3 = True
      |   if roundoverdistance == 0:
      |     findpoint3 = False
      |   end
      |   if findpoint3:
      |     # i need to find the point3 such that the arc from p2 to p3 to p4 is tangent to p1-p2 and p4-p5. making this a smooth path will be good
      |     # the direction of movement is from pointintersect in the direction of heading2
      |     # how much movement though? this will depend on whether it is actually a 90 degree angle or not.
      |     # first, find the perpendicular lines through points 2 and 4
      |     perp2 = find_perpendicular_line(ml1, point2[0], point2[1])
      |     perp4 = find_perpendicular_line(ml2, point4[0], point4[1])
      |     # next, find the intersection of those two lines
      |     perpintersect = find_intersection(perp2[0], perp2[1], perp4[0], perp4[1])
      |     radiusofcircle = distance_between(perpintersect[0], perpintersect[1], 0, point2[0], point2[1], 0)
      |     # find a vector the direction of heading2
      |     uvx = cos(heading2)
      |     uvy = sin(heading2)
      |     # compute point3. pass in negative radius because the direction is into the tank but we want to move from the intersection out to the rounded edge
      |     point3coords = add_vectordistance_to_point(perpintersect[0], perpintersect[1], z, uvx, uvy, 0, -1 * radiusofcircle)
      |     point3 = p[point3coords[0], point3coords[1], point3coords[2], 0, 0, 0]
      |   end
      | 
      |   #APPLY ACTUAL RXRYRZ TO POINTS
      |   # convert the headings to rxryrz and insert those values into the relevant points
      |   rxryrz = convert_heading_to_axang(heading1)
      |   rx = rxryrz[0]
      |   ry = rxryrz[1]
      |   rz = rxryrz[2]
      |   pointapproach1 = p[pointapproach1[0], pointapproach1[1], pointapproach1[2], rx, ry, rz]
      |   pointapproach2 = p[pointapproach2[0], pointapproach2[1], pointapproach2[2], rx, ry, rz]
      |   point1 = p[point1[0], point1[1], point1[2], rx, ry, rz]
      |   point2 = p[point2[0], point2[1], point2[2], rx, ry, rz]
      |   rxryrz = convert_heading_to_axang(heading2)
      |   rx = rxryrz[0]
      |   ry = rxryrz[1]
      |   rz = rxryrz[2]
      |   if findpoint3:
      |     point3 = p[point3[0], point3[1], point3[2], rx, ry, rz]
      |   else:
      |     point3 = point2
      |   end
      |   rxryrz = convert_heading_to_axang(heading3)
      |   rx = rxryrz[0]
      |   ry = rxryrz[1]
      |   rz = rxryrz[2]
      |   point4 = p[point4[0], point4[1], point4[2], rx, ry, rz]
      |   point5 = p[point5[0], point5[1], point5[2], rx, ry, rz]
      |   pointreturn1 = p[pointreturn1[0], pointreturn1[1], pointreturn1[2], rx, ry, rz]
      | 
      |   #find path2 (the part that goes up)
      |   four_vertical_points = find_vertical_points(pointintersect, l1delxunit, l1delyunit, l2delxunit, l2delyunit, zup, wd, heading1, heading3)
      |   path2r1 = four_vertical_points[0]
      |   path2r2 = four_vertical_points[1]
      |   path2l1 = four_vertical_points[2]
      |   path2l2 = four_vertical_points[3]
      | 
      |   #RETURN STRUCT
      |   ret = struct(pointintersect=pointintersect, pointapproach1=pointapproach1, pointapproach2=pointapproach2, point1=point1, point2=point2, point3=point3, point4=point4, point5=point5, pointreturn1=pointreturn1, heading1=heading1, heading2=heading2, heading3=heading3, path2r1=path2r1, path2r2=path2r2, path2l1=path2l1, path2l2=path2l2)
      |   return ret
      | end
      | 
      | # based on a Corner Homing 45 Cover pattern of touchpoints
      | # this uses those touchpoints to create a representation of the corner in 3d robot space.
      | def analyze_touchpoints_only_cover(p11, p12, p21, p3):
      |     zcoord=p3[2]
      | 
      |     # get the raw points from the first line
      |     l1p1x=p11[0]
      |     l1p1y=p11[1]
      |     l1p2x=p12[0]
      |     l1p2y=p12[1]
      | 
      |     # equate the first line in 2d space
      |     ml1 = (l1p2y-l1p1y) / (l1p2x-l1p1x)
      | 
      |     # b = y - mx
      |     bl1 = l1p1y - ml1 * l1p1x
      | 
      |     # get the raw points from the second line
      |     l2p1x=p21[0]
      |     l2p1y=p21[1]
      | 
      |     # equate the second line in 2d space
      |     # ml2 = opposite reciprocal of ml1 (because they are perpendicular) (assume perpendicular to make calculation of weldpath much easier)
      |     ml2 = -1 / ml1
      | 
      |     # b = y - mx
      |     bl2 = l2p1y - ml2 * l2p1x
      | 
      |     # find the intersection of the two lines
      |     # m1x+b1 = m2x+b2
      |     # m1x - m2x = b2 - b1
      |     # x = (b2-b1) / (m1-m2)
      |     xintersect = (bl2-bl1) / (ml1-ml2)
      |     yintersect = ml1 * xintersect + bl1
      | 
      |     pointintersect = p[xintersect,yintersect,zcoord,0,0,0]
      | 
      |     #FIND THE VECTORS
      |     #define a vector from the intersection to the second point on the first line
      |     l1delxfull = l1p2x - xintersect
      |     l1delyfull = l1p2y - yintersect
      | 
      |     l1delmag = sqrt(l1delxfull*l1delxfull + l1delyfull*l1delyfull)
      | 
      |     l1delxunit = l1delxfull / l1delmag
      |     l1delyunit = l1delyfull / l1delmag
      | 
      |     #define a vector from the intersection to the second point on the second line
      |     l2delxfull = l2p1x - xintersect
      |     l2delyfull = l2p1y - yintersect
      | 
      |     l2delmag = sqrt(l2delxfull*l2delxfull + l2delyfull*l2delyfull)
      | 
      |     l2delxunit = l2delxfull / l2delmag
      |     l2delyunit = l2delyfull / l2delmag
      | 
      |     #FIND HEADINGS
      |     #for each heading, find the angle of the line with respect to the pos x axis. this line is from pointintersect and along each edge of the corner
      |     heading1 = convert_uv_to_heading(l1delxunit, l1delyunit)
      |     heading3 = convert_uv_to_heading(l2delxunit, l2delyunit)
      |     # find halfway heading
      |     heading2 = (heading1 + heading3)/2
      | 
      |     #RETURN STRUCT
      |     ret = struct(pointintersect=pointintersect, heading1=heading1, heading2=heading2, heading3=heading3, l1delxunit=l1delxunit, l1delyunit=l1delyunit, l2delxunit=l2delxunit, l2delyunit=l2delyunit)
      |     return ret
      | end
      | 
      | # it takes 5 arguments as points
      | # it returns a struct containing: (pointintersect, heading1, heading2, heading3, l1delxunit, l1delyunit, l2delxunit, l2delyunit)
      | def analyze_touchpoints_only(p11, p12, p21, p22, p3):
      |   # FIND THE INTERSECTION
      |   # comment get the z
      |   zcoord=p3[2]
      | 
      |   # get the raw points from the first line
      |   l1p1x=p11[0]
      |   l1p1y=p11[1]
      |   l1p2x=p12[0]
      |   l1p2y=p12[1]
      | 
      |   # equate the first line in 2d space
      |   ml1 = (l1p2y-l1p1y) / (l1p2x-l1p1x)
      | 
      |   # b = y - mx
      |   bl1 = l1p1y - ml1 * l1p1x
      | 
      |   # get the raw points from the second line
      |   l2p1x=p21[0]
      |   l2p1y=p21[1]
      |   l2p2x=p22[0]
      |   l2p2y=p22[1]
      | 
      |   # equate the second line in 2d space
      |   ml2 = (l2p2y-l2p1y) / (l2p2x-l2p1x)
      | 
      |   # b = y - mx
      |   bl2 = l2p1y - ml2 * l2p1x
      | 
      | 
      |   # find the intersection of the two lines
      |   # m1x+b1 = m2x+b2
      |   # m1x - m2x = b2 - b1
      |   # x = (b2-b1) / (m1-m2)
      |   xintersect = (bl2-bl1) / (ml1-ml2)
      |   yintersect = ml1 * xintersect + bl1
      | 
      |   pointintersect = p[xintersect,yintersect,zcoord,0,0,0]
      | 
      |   #FIND THE VECTORS
      |   #define a vector from the intersection to the second point on the first line
      |   l1delxfull = l1p2x - xintersect
      |   l1delyfull = l1p2y - yintersect
      | 
      |   l1delmag = sqrt(l1delxfull*l1delxfull + l1delyfull*l1delyfull)
      | 
      |   l1delxunit = l1delxfull / l1delmag
      |   l1delyunit = l1delyfull / l1delmag
      | 
      |   #define a vector from the intersection to the second point on the second line
      |   l2delxfull = l2p2x - xintersect
      |   l2delyfull = l2p2y - yintersect
      | 
      |   l2delmag = sqrt(l2delxfull*l2delxfull + l2delyfull*l2delyfull)
      | 
      |   l2delxunit = l2delxfull / l2delmag
      |   l2delyunit = l2delyfull / l2delmag
      | 
      |   #FIND HEADINGS
      |   #for each heading, find the angle of the line with respect to the pos x axis. then add/subtract 90 degrees because you want to be perpendicular to that
      |   headingvector1 = convert_uv_to_heading(l1delxunit, l1delyunit)
      |   headingvector2 = convert_uv_to_heading(l2delxunit, l2delyunit)
      |   # find halfway heading
      |   heading2 = (headingvector1 + headingvector2)/2
      |   # find headings that the robot should face while traveling, perpendicular to the vectors of the sides of the box
